        (* Constant: '<S391>/Constant4' incorporates:
         *  Constant: '<S391>/Constant'
         *  Constant: '<S391>/Constant1'
         *  Constant: '<S391>/Constant2'
         *  Constant: '<S391>/Constant3' *)
        i3_Chart_Hysteresis_LowActive(ssMethodType := SS_INITIALIZE, sSignal := AI_DCHV_Plus_FB, boInitial_Value := FALSE, boValue_Activated := TRUE, boValue_Deactivated := FALSE, sLB := 5000.0, b_sUB := 10000.0);
        boOutput := i3_Chart_Hysteresis_LowActive.boOutput;
        (* SystemInitialize for Atomic SubSystem: '<Root>/ChiefMaster' *)
        (* SystemInitialize for Chart: '<S23>/Chart_DCPlus_Status' *)
        temporalCounter_i1_a(timerAction := 1, maxTime := 0);
        is_active_c54_ChiefMaster := 0;
        is_c54_ChiefMaster := ChiefMaster_IN_NO_ACTIVE_CHILD_f;
        (* SystemInitialize for Chart: '<S13>/delay1' *)
        temporalCounter_i1_h(timerAction := 1, maxTime := 0);
        is_active_c51_ChiefMaster := 0;
        is_c51_ChiefMaster := ChiefMaster_IN_NO_ACTIVE_CHILD_f;
        (* End of SystemInitialize for SubSystem: '<Root>/ChiefMaster' *)
        i0_InsulationMonitoringReq(ssMethodType := SS_INITIALIZE, IT_boUDC_KL15_D := rtb_IT_boUDC_KL15_D, IT_boUDC_KL15_C := rtb_IT_boUDC_KL15_C, IT_boBMS_HV_ON_BB := rtb_IT_boBMS_HV_ON_BB, IT_u8BMS_BB_No_MaxVoltage := rtb_Switch_a, IT_u8BMS_BB_No_MinVoltage := rtb_Switch2_k, IT_boBMS_SDError_BB1 := rtb_IT_boBMS_SDError_BB1, IT_boBMS_SDError_BB2 := rtb_IT_boBMS_SDError_BB1, IT_boBMS_SDError_BB3 := rtb_IT_boBMS_SDError_BB1, IT_boBMS_InsulationReadyOK_B1 := rtb_IT_boBMS_SDError_BB1, IT_boBMS_InsulationReadyOK_B2 := rtb_IT_boBMS_SDError_BB1, IT_boBMS_InsulationReadyOK_B3 := rtb_IT_boBMS_SDError_BB1, IT_boBMS_IMD_Active_BB1 := rtb_IT_boBMS_SDError_BB1, IT_boBMS_IMD_Active_BB2 := rtb_IT_boBMS_SDError_BB1, IT_boBMS_IMD_Active_BB3 := rtb_IT_boBMS_SDError_BB1, IT_boBMS_HV_REL_ON_BB1 := rtb_IT_boBMS_SDError_BB1, IT_boBMS_HV_REL_ON_BB2 := rtb_IT_boBMS_SDError_BB1, IT_boBMS_HV_REL_ON_BB3 := rtb_IT_boBMS_SDError_BB1, IT_sBMS_Batt1_Availability := DINT_TO_LREAL(rtb_UnitDelay5), IT_sBMS_Batt2_Availability := DINT_TO_LREAL(rtb_UnitDelay5), IT_sBMS_Batt3_Availability := DINT_TO_LREAL(rtb_UnitDelay5), IT_boUDC_EV_IsolationMeasurementRequest := rtb_IT_boUDC_EV_IsolationMeasurementRequest, FL_boSS_System_SD := System_Error, FL_boSS_System_ESD := rtb_Delay_j);
        rtb_IT_boChargeStop_Button := i0_InsulationMonitoringReq.FL_boREQ_IMD_ON_BB1;
        rtb_UnitDelay1_d := i0_InsulationMonitoringReq.FL_boREQ_IMD_ON_BB2;
        rtb_Out_bl := i0_InsulationMonitoringReq.FL_boREQ_IMD_ON_BB3;
        rtb_IMD_State_g := i0_InsulationMonitoringReq.FL_u8_IMD_State_BB1;
        rtb_System_SD_ErrorCode := i0_InsulationMonitoringReq.FL_u8_IMD_State_BB2;
        rtb_IMD_State := i0_InsulationMonitoringReq.FL_u8_IMD_State_BB3;
        (* Constant: '<S81>/Constant' *)
        i0_Chart_jj(ssMethodType := SS_INITIALIZE, In := ContactorState_f, b_n := 5.0);
        rtb_IT_boUDC_EV_IsolationMeasurementRequest := i0_Chart_jj.Out;
        i0_Chart1(ssMethodType := SS_INITIALIZE, In := rtb_IT_boBMS_SDError_BB1);
        rtb_Out_ap := i0_Chart1.Out;
        (* Constant: '<S82>/Constant' *)
        i1_Chart_jj(ssMethodType := SS_INITIALIZE, In := ContactorState, b_n := 5.0);
        rtb_IT_boUDC_EV_IsolationMeasurementRequest := i1_Chart_jj.Out;
        i1_Chart1(ssMethodType := SS_INITIALIZE, In := rtb_IT_boBMS_SDError_BB1);
        rtb_Out_ap := i1_Chart1.Out;
        i0_Chart_lg(ssMethodType := SS_INITIALIZE, Error := rtb_IT_boBMS_SDError_BB1, KL15_reset := rtb_IT_boBMS_SDError_BB1);
        rtb_IT_boUDC_EV_IsolationMeasurementRequest := i0_Chart_lg.SW_Reset;
        i0_Chart1_l(ssMethodType := SS_INITIALIZE, SW_Reset := rtb_IT_boUDC_EV_IsolationMeasurementRequest, KL_15_reset_CM := rtb_IT_boBMS_SDError_BB1);
        Count_k := i0_Chart1_l.Count;
        i1_Chart_lg(ssMethodType := SS_INITIALIZE, Error := rtb_IT_boBMS_SDError_BB1, KL15_reset := rtb_IT_boBMS_SDError_BB1);
        rtb_IT_boUDC_EV_IsolationMeasurementRequest := i1_Chart_lg.SW_Reset;
        i1_Chart1_l(ssMethodType := SS_INITIALIZE, SW_Reset := rtb_IT_boUDC_EV_IsolationMeasurementRequest, KL_15_reset_CM := rtb_IT_boBMS_SDError_BB1);
        Count_k := i1_Chart1_l.Count;
        i2_Chart_lg(ssMethodType := SS_INITIALIZE, Error := rtb_IT_boBMS_SDError_BB1, KL15_reset := rtb_IT_boBMS_SDError_BB1);
        rtb_IT_boUDC_EV_IsolationMeasurementRequest := i2_Chart_lg.SW_Reset;
        i2_Chart1_l(ssMethodType := SS_INITIALIZE, SW_Reset := rtb_IT_boUDC_EV_IsolationMeasurementRequest, KL_15_reset_CM := rtb_IT_boBMS_SDError_BB1);
        Count_k := i2_Chart1_l.Count;
        (* Constant: '<S86>/Constant' *)
        i2_Chart_jj(ssMethodType := SS_INITIALIZE, In := ContactorState_i, b_n := 5.0);
        rtb_IT_boUDC_EV_IsolationMeasurementRequest := i2_Chart_jj.Out;
        i2_Chart1(ssMethodType := SS_INITIALIZE, In := rtb_IT_boBMS_SDError_BB1);
        rtb_Out_ap := i2_Chart1.Out;
        i0_CMState(ssMethodType := SS_INITIALIZE, KL15 := rtb_IT_boBMS_SDError_BB1, KL15_AllBoxes := rtb_IT_boBMS_SDError_BB1, InsulationReadyOK := rtb_IT_boBMS_SDError_BB1, BattRelay_Closed := rtb_IT_boBMS_SDError_BB1, IMD_Available := rtb_IT_boBMS_SDError_BB1, BattRelay_Close_Req := rtb_IT_boBMS_SDError_BB1, REQ_IMD_ON := rtb_IT_boBMS_SDError_BB1, FL_boREQ_MainHV_ON_MINUS := rtb_IT_boBMS_SDError_BB1, MainHV_Plus_Status := DINT_TO_LREAL(rtb_UnitDelay5), ShutdownError := rtb_IT_boBMS_SDError_BB1);
        CMState_e2 := i0_CMState.FL_u8SS_ChiefMaster_State;
        (* Outport: '<Root>/DO_boEMSRET_BB1_1' *)
        i0_EMSRET_Power(ssMethodType := SS_INITIALIZE, ESD := rtb_Delay_j, HVILNOK := rtb_FL_boSS_HVIL_NOK, b_Reset := rtb_FL_boKL15_Reset);
        DO_boEMSRET_BB1_1 := i0_EMSRET_Power.FL_boSS_EMSRET_POWER;
        (* SystemInitialize for Atomic SubSystem: '<Root>/ChiefMaster' *)
        (* SystemInitialize for Chart: '<S108>/Chart' *)
        temporalCounter_i1(timerAction := 1, maxTime := 0);
        is_active_c49_ChiefMaster := 0;
        is_c49_ChiefMaster := ChiefMaster_IN_NO_ACTIVE_CHILD_f;
        (* End of SystemInitialize for SubSystem: '<Root>/ChiefMaster' *)
        

        (* ConstCode for Atomic SubSystem: '<Root>/ChiefMaster' *)
        (* ConstCode for ArithShift: '<S823>/Shift Arithmetic' incorporates:
         *  Constant: '<S803>/Constant' *)
        ShiftArithmetic := 0;
        (* ConstCode for ArithShift: '<S823>/Shift Arithmetic2' incorporates:
         *  Constant: '<S803>/Constant' *)
        ShiftArithmetic2 := 0;
        (* ConstCode for ArithShift: '<S823>/Shift Arithmetic4' incorporates:
         *  Constant: '<S803>/Constant' *)
        ShiftArithmetic4 := 0;
        (* ConstCode for ArithShift: '<S823>/Shift Arithmetic5' incorporates:
         *  Constant: '<S803>/Constant' *)
        ShiftArithmetic5 := 0;
        (* ConstCode for ArithShift: '<S823>/Shift Arithmetic6' incorporates:
         *  Constant: '<S803>/Constant' *)
        ShiftArithmetic6 := 0;
        (* ConstCode for ArithShift: '<S824>/Shift Arithmetic' incorporates:
         *  Constant: '<S803>/Constant2' *)
        ShiftArithmetic_n := 0;
        (* ConstCode for ArithShift: '<S824>/Shift Arithmetic2' incorporates:
         *  Constant: '<S803>/Constant2' *)
        ShiftArithmetic2_c := 0;
        (* ConstCode for ArithShift: '<S824>/Shift Arithmetic3' incorporates:
         *  Constant: '<S803>/Constant2' *)
        ShiftArithmetic3 := 0;
        (* ConstCode for ArithShift: '<S824>/Shift Arithmetic4' incorporates:
         *  Constant: '<S803>/Constant2' *)
        ShiftArithmetic4_h := 0;
        (* ConstCode for ArithShift: '<S824>/Shift Arithmetic5' incorporates:
         *  Constant: '<S803>/Constant2' *)
        ShiftArithmetic5_j := 0;
        (* ConstCode for ArithShift: '<S824>/Shift Arithmetic6' incorporates:
         *  Constant: '<S803>/Constant2' *)
        ShiftArithmetic6_a := 0;
        (* ConstCode for ArithShift: '<S825>/Shift Arithmetic6' incorporates:
         *  Constant: '<S803>/Constant' *)
        ShiftArithmetic6_f := 0;
        (* ConstCode for ArithShift: '<S860>/Shift Arithmetic2' incorporates:
         *  Constant: '<S804>/Constant4' *)
        ShiftArithmetic2_o := 0;
        (* ConstCode for ArithShift: '<S860>/Shift Arithmetic5' incorporates:
         *  Constant: '<S804>/Constant4' *)
        ShiftArithmetic5_h := 0;
        (* ConstCode for ArithShift: '<S898>/Shift Arithmetic2' incorporates:
         *  Constant: '<S807>/Constant4' *)
        ShiftArithmetic2_n := 0;
        (* ConstCode for ArithShift: '<S898>/Shift Arithmetic5' incorporates:
         *  Constant: '<S807>/Constant4' *)
        ShiftArithmetic5_jh := 0;
        (* ConstCode for ArithShift: '<S937>/Shift Arithmetic2' incorporates:
         *  Constant: '<S810>/Constant4' *)
        ShiftArithmetic2_h := 0;
        (* ConstCode for ArithShift: '<S937>/Shift Arithmetic5' incorporates:
         *  Constant: '<S810>/Constant4' *)
        ShiftArithmetic5_f := 0;
        (* ConstCode for ArithShift: '<S973>/Shift Arithmetic' incorporates:
         *  Constant: '<S813>/Constant' *)
        ShiftArithmetic_m := 0;
        (* ConstCode for ArithShift: '<S973>/Shift Arithmetic2' incorporates:
         *  Constant: '<S813>/Constant' *)
        ShiftArithmetic2_k := 0;
        (* ConstCode for ArithShift: '<S973>/Shift Arithmetic4' incorporates:
         *  Constant: '<S813>/Constant' *)
        ShiftArithmetic4_m := 0;
        (* ConstCode for ArithShift: '<S981>/Shift Arithmetic5' incorporates:
         *  Constant: '<S814>/Constant1' *)
        ShiftArithmetic5_k := 0;
        (* ConstCode for ArithShift: '<S981>/Shift Arithmetic6' incorporates:
         *  Constant: '<S814>/Constant1' *)
        ShiftArithmetic6_i := 0;
        (* ConstCode for ArithShift: '<S982>/Shift Arithmetic2' incorporates:
         *  Constant: '<S814>/Constant3' *)
        ShiftArithmetic2_p := 0;
        (* ConstCode for ArithShift: '<S982>/Shift Arithmetic3' incorporates:
         *  Constant: '<S814>/Constant3' *)
        ShiftArithmetic3_k := 0;
        (* ConstCode for ArithShift: '<S982>/Shift Arithmetic4' incorporates:
         *  Constant: '<S814>/Constant3' *)
        ShiftArithmetic4_a := 0;
        (* ConstCode for ArithShift: '<S982>/Shift Arithmetic5' incorporates:
         *  Constant: '<S814>/Constant3' *)
        ShiftArithmetic5_a := 0;
        (* ConstCode for ArithShift: '<S982>/Shift Arithmetic6' incorporates:
         *  Constant: '<S814>/Constant3' *)
        ShiftArithmetic6_m := 0;
        (* ConstCode for ArithShift: '<S991>/Shift Arithmetic2' incorporates:
         *  Constant: '<S815>/Constant4' *)
        ShiftArithmetic2_d := 0;
        (* ConstCode for ArithShift: '<S991>/Shift Arithmetic4' incorporates:
         *  Constant: '<S815>/Constant4' *)
        ShiftArithmetic4_n := 0;
        (* ConstCode for ArithShift: '<S991>/Shift Arithmetic6' incorporates:
         *  Constant: '<S815>/Constant4' *)
        ShiftArithmetic6_h := 0;
        (* ConstCode for ArithShift: '<S992>/Shift Arithmetic2' incorporates:
         *  Constant: '<S815>/Constant4' *)
        ShiftArithmetic2_b := 0;
        (* ConstCode for ArithShift: '<S992>/Shift Arithmetic3' incorporates:
         *  Constant: '<S815>/Constant4' *)
        ShiftArithmetic3_o := 0;
        (* ConstCode for ArithShift: '<S992>/Shift Arithmetic5' incorporates:
         *  Constant: '<S815>/Constant4' *)
        ShiftArithmetic5_a2 := 0;
        (* ConstCode for ArithShift: '<S992>/Shift Arithmetic6' incorporates:
         *  Constant: '<S815>/Constant4' *)
        ShiftArithmetic6_n := 0;
        (* ConstCode for ArithShift: '<S993>/Shift Arithmetic' incorporates:
         *  Constant: '<S815>/Constant1' *)
        ShiftArithmetic_h := 0;
        (* ConstCode for ArithShift: '<S993>/Shift Arithmetic1' incorporates:
         *  Constant: '<S815>/Constant1' *)
        ShiftArithmetic1 := 0;
        (* ConstCode for ArithShift: '<S993>/Shift Arithmetic3' incorporates:
         *  Constant: '<S815>/Constant1' *)
        ShiftArithmetic3_e := 0;
        (* ConstCode for ArithShift: '<S993>/Shift Arithmetic4' incorporates:
         *  Constant: '<S815>/Constant1' *)
        ShiftArithmetic4_ap := 0;
        (* ConstCode for ArithShift: '<S993>/Shift Arithmetic5' incorporates:
         *  Constant: '<S815>/Constant1' *)
        ShiftArithmetic5_i := 0;
        (* ConstCode for ArithShift: '<S993>/Shift Arithmetic6' incorporates:
         *  Constant: '<S815>/Constant1' *)
        ShiftArithmetic6_k := 0;
        (* ConstCode for DataTypeConversion: '<S1020>/Data Type Conversion1' incorporates:
         *  Constant: '<S1017>/Constant15' *)
        DataTypeConversion1 := 0;
        (* ConstCode for DataTypeConversion: '<S1020>/Data Type Conversion2' incorporates:
         *  Constant: '<S1017>/Constant15' *)
        DataTypeConversion2 := 0;
        (* ConstCode for DataTypeConversion: '<S1020>/Data Type Conversion4' incorporates:
         *  Constant: '<S1017>/Constant15' *)
        DataTypeConversion4 := 0;
        (* ConstCode for DataTypeConversion: '<S1020>/Data Type Conversion5' incorporates:
         *  Constant: '<S1017>/Constant15' *)
        DataTypeConversion5 := 0;
        (* ConstCode for DataTypeConversion: '<S1020>/Data Type Conversion6' incorporates:
         *  Constant: '<S1017>/Constant15' *)
        DataTypeConversion6 := 0;
        (* ConstCode for DataTypeConversion: '<S1020>/Data Type Conversion7' incorporates:
         *  Constant: '<S1017>/Constant15' *)
        DataTypeConversion7 := 0;
        (* ConstCode for ArithShift: '<S1020>/Shift Arithmetic1' incorporates:
         *  DataTypeConversion: '<S1020>/Data Type Conversion1' *)
        ShiftArithmetic1_n := BYTE_TO_USINT(SHL(USINT_TO_BYTE(DataTypeConversion1), 2));
        (* ConstCode for ArithShift: '<S1020>/Shift Arithmetic2' incorporates:
         *  DataTypeConversion: '<S1020>/Data Type Conversion2' *)
        ShiftArithmetic2_ot := BYTE_TO_USINT(SHL(USINT_TO_BYTE(DataTypeConversion2), 3));
        (* ConstCode for ArithShift: '<S1020>/Shift Arithmetic3' incorporates:
         *  DataTypeConversion: '<S1020>/Data Type Conversion4' *)
        ShiftArithmetic3_oe := BYTE_TO_USINT(SHL(USINT_TO_BYTE(DataTypeConversion4), 4));
        (* ConstCode for ArithShift: '<S1020>/Shift Arithmetic4' incorporates:
         *  DataTypeConversion: '<S1020>/Data Type Conversion5' *)
        ShiftArithmetic4_d := BYTE_TO_USINT(SHL(USINT_TO_BYTE(DataTypeConversion5), 5));
        (* ConstCode for ArithShift: '<S1020>/Shift Arithmetic5' incorporates:
         *  DataTypeConversion: '<S1020>/Data Type Conversion6' *)
        ShiftArithmetic5_ke := BYTE_TO_USINT(SHL(USINT_TO_BYTE(DataTypeConversion6), 6));
        (* ConstCode for ArithShift: '<S1020>/Shift Arithmetic6' incorporates:
         *  DataTypeConversion: '<S1020>/Data Type Conversion7' *)
        ShiftArithmetic6_kx := BYTE_TO_USINT(SHL(USINT_TO_BYTE(DataTypeConversion7), 7));
        (* ConstCode for DataTypeConversion: '<S1021>/Data Type Conversion1' incorporates:
         *  Constant: '<S1018>/Constant1' *)
        DataTypeConversion1_l := 0;
        (* ConstCode for DataTypeConversion: '<S1021>/Data Type Conversion2' incorporates:
         *  Constant: '<S1018>/Constant1' *)
        DataTypeConversion2_b := 0;
        (* ConstCode for DataTypeConversion: '<S1021>/Data Type Conversion4' incorporates:
         *  Constant: '<S1018>/Constant1' *)
        DataTypeConversion4_l := 0;
        (* ConstCode for DataTypeConversion: '<S1021>/Data Type Conversion5' incorporates:
         *  Constant: '<S1018>/Constant1' *)
        DataTypeConversion5_k := 0;
        (* ConstCode for DataTypeConversion: '<S1021>/Data Type Conversion6' incorporates:
         *  Constant: '<S1018>/Constant1' *)
        DataTypeConversion6_e := 0;
        (* ConstCode for DataTypeConversion: '<S1021>/Data Type Conversion7' incorporates:
         *  Constant: '<S1018>/Constant1' *)
        DataTypeConversion7_p := 0;
        (* ConstCode for ArithShift: '<S1021>/Shift Arithmetic1' incorporates:
         *  DataTypeConversion: '<S1021>/Data Type Conversion1' *)
        ShiftArithmetic1_nm := BYTE_TO_USINT(SHL(USINT_TO_BYTE(DataTypeConversion1_l), 2));
        (* ConstCode for ArithShift: '<S1021>/Shift Arithmetic2' incorporates:
         *  DataTypeConversion: '<S1021>/Data Type Conversion2' *)
        ShiftArithmetic2_e := BYTE_TO_USINT(SHL(USINT_TO_BYTE(DataTypeConversion2_b), 3));
        (* ConstCode for ArithShift: '<S1021>/Shift Arithmetic3' incorporates:
         *  DataTypeConversion: '<S1021>/Data Type Conversion4' *)
        ShiftArithmetic3_o0 := BYTE_TO_USINT(SHL(USINT_TO_BYTE(DataTypeConversion4_l), 4));
        (* ConstCode for ArithShift: '<S1021>/Shift Arithmetic4' incorporates:
         *  DataTypeConversion: '<S1021>/Data Type Conversion5' *)
        ShiftArithmetic4_b := BYTE_TO_USINT(SHL(USINT_TO_BYTE(DataTypeConversion5_k), 5));
        (* ConstCode for ArithShift: '<S1021>/Shift Arithmetic5' incorporates:
         *  DataTypeConversion: '<S1021>/Data Type Conversion6' *)
        ShiftArithmetic5_hi := BYTE_TO_USINT(SHL(USINT_TO_BYTE(DataTypeConversion6_e), 6));
        (* ConstCode for ArithShift: '<S1021>/Shift Arithmetic6' incorporates:
         *  DataTypeConversion: '<S1021>/Data Type Conversion7' *)
        ShiftArithmetic6_kxt := BYTE_TO_USINT(SHL(USINT_TO_BYTE(DataTypeConversion7_p), 7));
        (* ConstCode for DataTypeConversion: '<S1022>/Data Type Conversion1' incorporates:
         *  Constant: '<S1019>/Constant2' *)
        DataTypeConversion1_o := 0;
        (* ConstCode for DataTypeConversion: '<S1022>/Data Type Conversion2' incorporates:
         *  Constant: '<S1019>/Constant2' *)
        DataTypeConversion2_o := 0;
        (* ConstCode for DataTypeConversion: '<S1022>/Data Type Conversion4' incorporates:
         *  Constant: '<S1019>/Constant2' *)
        DataTypeConversion4_i := 0;
        (* ConstCode for DataTypeConversion: '<S1022>/Data Type Conversion5' incorporates:
         *  Constant: '<S1019>/Constant2' *)
        DataTypeConversion5_n := 0;
        (* ConstCode for DataTypeConversion: '<S1022>/Data Type Conversion6' incorporates:
         *  Constant: '<S1019>/Constant2' *)
        DataTypeConversion6_k := 0;
        (* ConstCode for DataTypeConversion: '<S1022>/Data Type Conversion7' incorporates:
         *  Constant: '<S1019>/Constant2' *)
        DataTypeConversion7_pe := 0;
        (* ConstCode for ArithShift: '<S1022>/Shift Arithmetic1' incorporates:
         *  DataTypeConversion: '<S1022>/Data Type Conversion1' *)
        ShiftArithmetic1_nx := BYTE_TO_USINT(SHL(USINT_TO_BYTE(DataTypeConversion1_o), 2));
        (* ConstCode for ArithShift: '<S1022>/Shift Arithmetic2' incorporates:
         *  DataTypeConversion: '<S1022>/Data Type Conversion2' *)
        ShiftArithmetic2_m := BYTE_TO_USINT(SHL(USINT_TO_BYTE(DataTypeConversion2_o), 3));
        (* ConstCode for ArithShift: '<S1022>/Shift Arithmetic3' incorporates:
         *  DataTypeConversion: '<S1022>/Data Type Conversion4' *)
        ShiftArithmetic3_a := BYTE_TO_USINT(SHL(USINT_TO_BYTE(DataTypeConversion4_i), 4));
        (* ConstCode for ArithShift: '<S1022>/Shift Arithmetic4' incorporates:
         *  DataTypeConversion: '<S1022>/Data Type Conversion5' *)
        ShiftArithmetic4_p := BYTE_TO_USINT(SHL(USINT_TO_BYTE(DataTypeConversion5_n), 5));
        (* ConstCode for ArithShift: '<S1022>/Shift Arithmetic5' incorporates:
         *  DataTypeConversion: '<S1022>/Data Type Conversion6' *)
        ShiftArithmetic5_b := BYTE_TO_USINT(SHL(USINT_TO_BYTE(DataTypeConversion6_k), 6));
        (* ConstCode for ArithShift: '<S1022>/Shift Arithmetic6' incorporates:
         *  DataTypeConversion: '<S1022>/Data Type Conversion7' *)
        ShiftArithmetic6_b := BYTE_TO_USINT(SHL(USINT_TO_BYTE(DataTypeConversion7_pe), 7));
        (* ConstCode for DataTypeConversion: '<S1026>/Extract Desired Bits' incorporates:
         *  Constant: '<S1023>/Constant4' *)
        ExtractDesiredBits := 0;
        (* ConstCode for DataTypeConversion: '<S1028>/Extract Desired Bits' incorporates:
         *  Constant: '<S1023>/Constant5' *)
        ExtractDesiredBits_m := 1;
        (* ConstCode for DataTypeConversion: '<S1031>/Data Type Conversion3' incorporates:
         *  DataTypeConversion: '<S1026>/Extract Desired Bits' *)
        DataTypeConversion3 := ExtractDesiredBits;
        (* ConstCode for DataTypeConversion: '<S1031>/Data Type Conversion6' incorporates:
         *  DataTypeConversion: '<S1028>/Extract Desired Bits' *)
        DataTypeConversion6_h := ExtractDesiredBits_m;
        (* ConstCode for ArithShift: '<S1031>/Shift Arithmetic' incorporates:
         *  Constant: '<S1023>/Constant1' *)
        ShiftArithmetic_k := 0;
        (* ConstCode for ArithShift: '<S1031>/Shift Arithmetic2' incorporates:
         *  Constant: '<S1023>/Constant2' *)
        ShiftArithmetic2_f := 0;
        (* ConstCode for ArithShift: '<S1031>/Shift Arithmetic3' incorporates:
         *  Constant: '<S1023>/Constant2' *)
        ShiftArithmetic3_h := 0;
        (* ConstCode for ArithShift: '<S1031>/Shift Arithmetic4' incorporates:
         *  Constant: '<S1023>/Constant2' *)
        ShiftArithmetic4_l := 0;
        (* ConstCode for ArithShift: '<S1031>/Shift Arithmetic5' incorporates:
         *  DataTypeConversion: '<S1031>/Data Type Conversion6' *)
        ShiftArithmetic5_m := BYTE_TO_USINT(SHL(USINT_TO_BYTE(DataTypeConversion6_h), 6));
        (* ConstCode for ArithShift: '<S1031>/Shift Arithmetic6' incorporates:
         *  Constant: '<S1023>/Constant3' *)
        ShiftArithmetic6_ap := 0;
        (* ConstCode for DataTypeConversion: '<S1032>/Extract Desired Bits' incorporates:
         *  Constant: '<S1024>/Constant4' *)
        ExtractDesiredBits_n := 0;
        (* ConstCode for DataTypeConversion: '<S1034>/Extract Desired Bits' incorporates:
         *  Constant: '<S1024>/Constant5' *)
        ExtractDesiredBits_b := 1;
        (* ConstCode for DataTypeConversion: '<S1037>/Data Type Conversion3' incorporates:
         *  DataTypeConversion: '<S1032>/Extract Desired Bits' *)
        DataTypeConversion3_d := ExtractDesiredBits_n;
        (* ConstCode for DataTypeConversion: '<S1037>/Data Type Conversion6' incorporates:
         *  DataTypeConversion: '<S1034>/Extract Desired Bits' *)
        DataTypeConversion6_p := ExtractDesiredBits_b;
        (* ConstCode for ArithShift: '<S1037>/Shift Arithmetic' incorporates:
         *  Constant: '<S1024>/Constant1' *)
        ShiftArithmetic_a := 0;
        (* ConstCode for ArithShift: '<S1037>/Shift Arithmetic2' incorporates:
         *  Constant: '<S1024>/Constant2' *)
        ShiftArithmetic2_fl := 0;
        (* ConstCode for ArithShift: '<S1037>/Shift Arithmetic3' incorporates:
         *  Constant: '<S1024>/Constant2' *)
        ShiftArithmetic3_l := 0;
        (* ConstCode for ArithShift: '<S1037>/Shift Arithmetic4' incorporates:
         *  Constant: '<S1024>/Constant2' *)
        ShiftArithmetic4_f := 0;
        (* ConstCode for ArithShift: '<S1037>/Shift Arithmetic5' incorporates:
         *  DataTypeConversion: '<S1037>/Data Type Conversion6' *)
        ShiftArithmetic5_k0 := BYTE_TO_USINT(SHL(USINT_TO_BYTE(DataTypeConversion6_p), 6));
        (* ConstCode for ArithShift: '<S1037>/Shift Arithmetic6' incorporates:
         *  Constant: '<S1024>/Constant3' *)
        ShiftArithmetic6_o := 0;
        (* ConstCode for DataTypeConversion: '<S1038>/Extract Desired Bits' incorporates:
         *  Constant: '<S1025>/Constant4' *)
        ExtractDesiredBits_m1 := 0;
        (* ConstCode for DataTypeConversion: '<S1040>/Extract Desired Bits' incorporates:
         *  Constant: '<S1025>/Constant5' *)
        ExtractDesiredBits_p := 1;
        (* ConstCode for DataTypeConversion: '<S1043>/Data Type Conversion3' incorporates:
         *  DataTypeConversion: '<S1038>/Extract Desired Bits' *)
        DataTypeConversion3_l := ExtractDesiredBits_m1;
        (* ConstCode for DataTypeConversion: '<S1043>/Data Type Conversion6' incorporates:
         *  DataTypeConversion: '<S1040>/Extract Desired Bits' *)
        DataTypeConversion6_l := ExtractDesiredBits_p;
        (* ConstCode for ArithShift: '<S1043>/Shift Arithmetic' incorporates:
         *  Constant: '<S1025>/Constant1' *)
        ShiftArithmetic_p := 0;
        (* ConstCode for ArithShift: '<S1043>/Shift Arithmetic2' incorporates:
         *  Constant: '<S1025>/Constant2' *)
        ShiftArithmetic2_g := 0;
        (* ConstCode for ArithShift: '<S1043>/Shift Arithmetic3' incorporates:
         *  Constant: '<S1025>/Constant2' *)
        ShiftArithmetic3_c := 0;
        (* ConstCode for ArithShift: '<S1043>/Shift Arithmetic4' incorporates:
         *  Constant: '<S1025>/Constant2' *)
        ShiftArithmetic4_db := 0;
        (* ConstCode for ArithShift: '<S1043>/Shift Arithmetic5' incorporates:
         *  DataTypeConversion: '<S1043>/Data Type Conversion6' *)
        ShiftArithmetic5_c := BYTE_TO_USINT(SHL(USINT_TO_BYTE(DataTypeConversion6_l), 6));
        (* ConstCode for ArithShift: '<S1043>/Shift Arithmetic6' incorporates:
         *  Constant: '<S1025>/Constant3' *)
        ShiftArithmetic6_mw := 0;
        (* End of ConstCode for SubSystem: '<Root>/ChiefMaster' *)
    SS_STEP: 
        (* Outputs for Atomic SubSystem: '<Root>/ChiefMaster' *)
        (* Outputs for Enabled SubSystem: '<S195>/Subsystem1' incorporates:
         *  EnablePort: '<S664>/Timeout' *)
        (* Logic: '<S195>/NOT' *)

        IF  NOT C_UDC_Msg1_Timeout THEN 

            IF  NOT Subsystem1_MODE THEN 
                Subsystem1_MODE := TRUE;
            END_IF;

            (* DataTypeConversion: '<S664>/Data Type Conversion2' incorporates:
             *  DataTypeConversion: '<S666>/Extract Desired Bits' *)
            IP_boSafeToShutdown := DWORD_TO_UDINT(UDINT_TO_DWORD(USINT_TO_UDINT(C_UDC_Msg1[0])) AND 1) <> 0;
            (* DataTypeConversion: '<S664>/Data Type Conversion3' incorporates:
             *  DataTypeConversion: '<S667>/Extract Desired Bits' *)
            IP_boKL15_D := DWORD_TO_UDINT(UDINT_TO_DWORD(DINT_TO_UDINT(DWORD_TO_DINT(SHR(DINT_TO_DWORD(USINT_TO_DINT(C_UDC_Msg1[0])), 1)))) AND 1) <> 0;
            (* DataTypeConversion: '<S664>/Data Type Conversion4' incorporates:
             *  DataTypeConversion: '<S668>/Extract Desired Bits' *)
            IP_boKL15_C := DWORD_TO_UDINT(UDINT_TO_DWORD(DINT_TO_UDINT(DWORD_TO_DINT(SHR(DINT_TO_DWORD(USINT_TO_DINT(C_UDC_Msg1[0])), 2)))) AND 1) <> 0;
            (* DataTypeConversion: '<S664>/Data Type Conversion5' incorporates:
             *  DataTypeConversion: '<S669>/Extract Desired Bits' *)
            IP_boEVDisconnectingDevice := DWORD_TO_UDINT(UDINT_TO_DWORD(DINT_TO_UDINT(DWORD_TO_DINT(SHR(DINT_TO_DWORD(USINT_TO_DINT(C_UDC_Msg1[0])), 3)))) AND 1) <> 0;
            (* DataTypeConversion: '<S664>/Data Type Conversion7' incorporates:
             *  DataTypeConversion: '<S671>/Extract Desired Bits' *)
            IP_boChargeStop_Button := DWORD_TO_UDINT(UDINT_TO_DWORD(DINT_TO_UDINT(DWORD_TO_DINT(SHR(DINT_TO_DWORD(USINT_TO_DINT(C_UDC_Msg1[0])), 5)))) AND 1) <> 0;
            (* SignalConversion: '<S664>/TmpBufferAtConstantOutport1' incorporates:
             *  Constant: '<S664>/Constant' *)
            IP_boEV_IsolationMeasurementRequest := TRUE;
        ELSIF Subsystem1_MODE THEN 
            (* Disable for DataTypeConversion: '<S664>/Data Type Conversion2' incorporates:
             *  Outport: '<S664>/TTC_Status_Databus' *)
            IP_boSafeToShutdown := FALSE;
            (* Disable for DataTypeConversion: '<S664>/Data Type Conversion3' incorporates:
             *  Outport: '<S664>/TTC_Status_Databus' *)
            IP_boKL15_D := FALSE;
            (* Disable for DataTypeConversion: '<S664>/Data Type Conversion4' incorporates:
             *  Outport: '<S664>/TTC_Status_Databus' *)
            IP_boKL15_C := FALSE;
            (* Disable for DataTypeConversion: '<S664>/Data Type Conversion5' incorporates:
             *  Outport: '<S664>/TTC_Status_Databus' *)
            IP_boEVDisconnectingDevice := FALSE;
            (* Disable for SignalConversion: '<S664>/TmpBufferAtConstantOutport1' incorporates:
             *  Outport: '<S664>/TTC_Status_Databus' *)
            IP_boEV_IsolationMeasurementRequest := FALSE;
            (* Disable for DataTypeConversion: '<S664>/Data Type Conversion7' incorporates:
             *  Outport: '<S664>/TTC_Status_Databus' *)
            IP_boChargeStop_Button := FALSE;
            Subsystem1_MODE := FALSE;
        END_IF;

        (* End of Logic: '<S195>/NOT' *)
        (* End of Outputs for SubSystem: '<S195>/Subsystem1' *)
        

        (* SignalConversion: '<S678>/Signal Copy5' *)
        rtb_IT_boUDC_EV_IsolationMeasurementRequest := IP_boEV_IsolationMeasurementRequest;
        (* SignalConversion: '<S678>/Signal Copy6' *)
        rtb_IT_boChargeStop_Button := IP_boChargeStop_Button;
        (* End of Outputs for SubSystem: '<Root>/ChiefMaster' *)
        

        (* Constant: '<S387>/Constant4' incorporates:
         *  Constant: '<S387>/Constant'
         *  Constant: '<S387>/Constant1'
         *  Constant: '<S387>/Constant2'
         *  Constant: '<S387>/Constant3' *)
        i5_Chart_Hysteresis_HighActive(ssMethodType := SS_OUTPUT, sSignal := AI_KL15, boInitial_Value := FALSE, boValue_Activated := TRUE, boValue_Deactivated := FALSE, sLB := 18000.0, b_sUB := 22000.0);
        boOutput_c := i5_Chart_Hysteresis_HighActive.boOutput;
        (* Outputs for Atomic SubSystem: '<Root>/ChiefMaster' *)
        (* SignalConversion: '<S677>/Signal Copy' *)
        rtb_IT_boBMS_SDError_BB1 := boOutput_c;
        (* Logic: '<S55>/NOT1' incorporates:
         *  RelationalOperator: '<S61>/Compare'
         *  SignalConversion: '<S677>/Signal Copy' *)
        rtb_S_in :=  NOT boOutput_c;
        (* Logic: '<S56>/NOT' incorporates:
         *  Constant: '<S60>/Constant'
         *  Constant: '<S62>/Constant'
         *  Constant: '<S63>/Constant'
         *  Logic: '<S56>/OR'
         *  Logic: '<S56>/OR1'
         *  Logic: '<S56>/OR2'
         *  Outport: '<Root>/DO_KL15_BB1'
         *  RelationalOperator: '<S60>/Compare'
         *  RelationalOperator: '<S62>/Compare'
         *  RelationalOperator: '<S63>/Compare'
         *  UnitDelay: '<S10>/Unit Delay'
         *  UnitDelay: '<S10>/Unit Delay6' *)
        i0_Chart_m(ssMethodType := SS_OUTPUT, In := (( NOT rtb_S_in) AND (UnitDelay_DSTATE <> 1.0)) OR ((UnitDelay6_DSTATE <> 1.0) AND (UnitDelay6_DSTATE <> 3.0)), KL15_CM_Reset := rtb_S_in);
        DO_KL15_BB1 := i0_Chart_m.Out;
        (* RelationalOperator: '<S66>/Compare' incorporates:
         *  Logic: '<S55>/NOR'
         *  RelationalOperator: '<S71>/Compare' *)
        rtb_out_n :=  NOT rtb_IT_boBMS_SDError_BB1;
        (* Logic: '<S57>/NOT' incorporates:
         *  Constant: '<S65>/Constant'
         *  Constant: '<S67>/Constant'
         *  Constant: '<S68>/Constant'
         *  Logic: '<S57>/OR'
         *  Logic: '<S57>/OR1'
         *  Logic: '<S57>/OR2'
         *  Outport: '<Root>/DO_KL15_BB2'
         *  RelationalOperator: '<S65>/Compare'
         *  RelationalOperator: '<S66>/Compare'
         *  RelationalOperator: '<S67>/Compare'
         *  RelationalOperator: '<S68>/Compare'
         *  UnitDelay: '<S10>/Unit Delay1'
         *  UnitDelay: '<S10>/Unit Delay7' *)
        i1_Chart_m(ssMethodType := SS_OUTPUT, In := (( NOT rtb_out_n) AND (UnitDelay1_DSTATE <> 1.0)) OR ((UnitDelay7_DSTATE <> 1.0) AND (UnitDelay7_DSTATE <> 3.0)), KL15_CM_Reset := rtb_out_n);
        DO_KL15_BB2 := i1_Chart_m.Out;
        (* Logic: '<S58>/NOT' incorporates:
         *  Constant: '<S70>/Constant'
         *  Constant: '<S72>/Constant'
         *  Constant: '<S73>/Constant'
         *  Logic: '<S58>/OR'
         *  Logic: '<S58>/OR1'
         *  Logic: '<S58>/OR2'
         *  Outport: '<Root>/DO_KL15_BB3'
         *  RelationalOperator: '<S70>/Compare'
         *  RelationalOperator: '<S72>/Compare'
         *  RelationalOperator: '<S73>/Compare'
         *  UnitDelay: '<S10>/Unit Delay2'
         *  UnitDelay: '<S10>/Unit Delay8' *)
        i2_Chart_m(ssMethodType := SS_OUTPUT, In := (( NOT rtb_out_n) AND (UnitDelay2_DSTATE <> 1.0)) OR ((UnitDelay8_DSTATE <> 1.0) AND (UnitDelay8_DSTATE <> 3.0)), KL15_CM_Reset := rtb_out_n);
        DO_KL15_BB3 := i2_Chart_m.Out;
        (* Logic: '<S55>/AND' incorporates:
         *  Logic: '<S55>/NOT1'
         *  Logic: '<S55>/NOT2'
         *  Logic: '<S55>/NOT3'
         *  Logic: '<S55>/NOT4'
         *  Outport: '<Root>/DO_KL15_BB1'
         *  Outport: '<Root>/DO_KL15_BB2'
         *  Outport: '<Root>/DO_KL15_BB3' *)
        rtb_FL_boCMSleep := ((rtb_S_in AND ( NOT DO_KL15_BB1)) AND ( NOT DO_KL15_BB2)) AND ( NOT DO_KL15_BB3);
        (* SignalConversion: '<S678>/Signal Copy1' *)
        rtb_IT_boUDC_KL15_D := IP_boKL15_D;
        (* SignalConversion: '<S678>/Signal Copy2' *)
        rtb_IT_boUDC_KL15_C := IP_boKL15_C;
        (* Logic: '<S55>/AND6' incorporates:
         *  SignalConversion: '<S678>/Signal Copy1'
         *  SignalConversion: '<S678>/Signal Copy2' *)
        rtb_FL_boKL15_Disable := IP_boKL15_D = IP_boKL15_C;
        (* Switch: '<S431>/Switch' incorporates:
         *  Constant: '<S431>/Constant'
         *  Constant: '<S431>/Constant1'
         *  Logic: '<S431>/AND'
         *  Logic: '<S431>/NOT'
         *  Logic: '<S431>/NOT1'
         *  Logic: '<S431>/NOT2'
         *  Logic: '<S431>/NOT3'
         *  Logic: '<S431>/NOT4'
         *  Logic: '<S431>/NOT5'
         *  Logic: '<S431>/NOT6' *)

        IF (((((( NOT C_LB_Batt1_CellVoltage01_Timeout) AND ( NOT C_LB_Batt1_CellVoltage02_Timeout)) AND ( NOT C_LB_Batt1_CellTemperature_Timeout)) AND ( NOT C_LB_Batt1_InsulationMonitor_Timeout)) AND ( NOT C_LB_Batt1_Status01_Timeout)) AND ( NOT C_LB_Batt1_Status02_Timeout)) AND ( NOT C_LB_Batt1_Status03_Timeout) THEN 
            rtb_Switch2_d := TRUE;
            (* Switch: '<S675>/Switch1' incorporates:
             *  Constant: '<S431>/Constant'
             *  Constant: '<S675>/Constant6' *)
            rtb_S_in := TRUE;
        ELSE 
            rtb_Switch2_d := FALSE;
            (* Switch: '<S675>/Switch1' incorporates:
             *  Constant: '<S431>/Constant1'
             *  Constant: '<S675>/Constant7' *)
            rtb_S_in := FALSE;
        END_IF;

        (* End of Switch: '<S431>/Switch' *)
        

        (* Switch: '<S200>/Switch' incorporates:
         *  Logic: '<S200>/AND'
         *  Logic: '<S200>/NOT'
         *  Logic: '<S200>/NOT1'
         *  Logic: '<S200>/NOT2'
         *  Logic: '<S200>/NOT3'
         *  Logic: '<S200>/NOT4'
         *  Logic: '<S200>/NOT5' *)

        IF ((((( NOT C_Actia_Batt1_MyStatus_Timeout) AND ( NOT C_Actia_Batt1_Error_Timeout)) AND ( NOT C_Actia_Batt1_ADS_8_Timeout)) AND ( NOT C_Actia_Batt1_ADS_0_Timeout)) AND ( NOT C_Actia_Batt1_ADS_1_Timeout)) AND ( NOT C_Actia_Batt1_ADS_3_Timeout) THEN 
            (* Switch: '<S675>/Switch' incorporates:
             *  Constant: '<S675>/Constant3' *)
            rtb_IP_boBatt1_Actia_Availability := TRUE;
        ELSE 
            (* Switch: '<S675>/Switch' incorporates:
             *  Constant: '<S675>/Constant4' *)
            rtb_IP_boBatt1_Actia_Availability := FALSE;
        END_IF;

        (* End of Switch: '<S200>/Switch' *)
        (* End of Outputs for SubSystem: '<Root>/ChiefMaster' *)
        i0_ChartBatt1(ssMethodType := SS_OUTPUT, BattAvailable_LiBa := rtb_S_in, BattAvailable_Actia := rtb_IP_boBatt1_Actia_Availability);
        rtb_BattSelect_f := i0_ChartBatt1.BattSelect;
        (* Outputs for Atomic SubSystem: '<Root>/ChiefMaster' *)
        (* Sum: '<S208>/Add' incorporates:
         *  ArithShift: '<S207>/Shift Arithmetic'
         *  Constant: '<S206>/Constant'
         *  DataTypeConversion: '<S207>/Data Type Conversion'
         *  Product: '<S208>/Product'
         *  Sum: '<S207>/Add' *)
        rtb_Min := DINT_TO_REAL(DWORD_TO_DINT(SHL(DINT_TO_DWORD(USINT_TO_DINT(C_Actia_Batt1_ADS_3[2])), 8)) + USINT_TO_DINT(C_Actia_Batt1_ADS_3[1])) * 0.1;
        (* Sum: '<S498>/Add' incorporates:
         *  ArithShift: '<S497>/Shift Arithmetic'
         *  Constant: '<S493>/Constant'
         *  DataTypeConversion: '<S497>/Data Type Conversion'
         *  Product: '<S498>/Product'
         *  Sum: '<S497>/Add' *)
        rtb_Add_psl := DINT_TO_REAL(DWORD_TO_DINT(SHL(DINT_TO_DWORD(USINT_TO_DINT(C_LB_BMS_Status02_Msg[7])), 8)) + USINT_TO_DINT(C_LB_BMS_Status02_Msg[6])) * 0.1;
        (* Switch: '<S498>/Switch' incorporates:
         *  Constant: '<S493>/Constant3'
         *  Constant: '<S493>/Constant4'
         *  RelationalOperator: '<S498>/GreaterThan'
         *  Switch: '<S498>/Switch1' *)

        IF C_LB_Batt1_Status02_Timeout THEN 
            rtb_Add_psl := 0.0;
        ELSIF rtb_Add_psl > 6553.5 THEN 
            (* Switch: '<S498>/Switch1' incorporates:
             *  Constant: '<S493>/Constant4' *)
            rtb_Add_psl := 0.0;
        END_IF;

        (* End of Switch: '<S498>/Switch' *)
        

        (* MultiPortSwitch: '<S712>/Multiport Switch' incorporates:
         *  Constant: '<S712>/Constant' *)

        CASE TRUNC(rtb_BattSelect_f) OF
            1: 
                (* Switch: '<S208>/Switch' incorporates:
                 *  Constant: '<S206>/Constant3'
                 *  Constant: '<S206>/SafeValue_NA '
                 *  RelationalOperator: '<S208>/GreaterThan'
                 *  Switch: '<S208>/Switch1' *)

                IF C_Actia_Batt1_ADS_3_Timeout THEN 
                    rtb_Min := 0.0;
                ELSIF rtb_Min > 6553.5 THEN 
                    (* Switch: '<S208>/Switch1' incorporates:
                     *  Constant: '<S206>/SafeValue_Error' *)
                    rtb_Min := 0.0;
                END_IF;

                (* End of Switch: '<S208>/Switch' *)
            2: 
                rtb_Min := rtb_Add_psl;
            3: 
                rtb_Min := 0.0;
            ELSE
                rtb_Min := 0.0;
        END_CASE;

        (* End of MultiPortSwitch: '<S712>/Multiport Switch' *)
        

        (* Switch: '<S511>/Switch' incorporates:
         *  Constant: '<S511>/Constant'
         *  Constant: '<S511>/Constant1'
         *  Logic: '<S511>/AND'
         *  Logic: '<S511>/NOT'
         *  Logic: '<S511>/NOT1'
         *  Logic: '<S511>/NOT2'
         *  Logic: '<S511>/NOT3'
         *  Logic: '<S511>/NOT4'
         *  Logic: '<S511>/NOT5'
         *  Logic: '<S511>/NOT6' *)

        IF (((((( NOT C_LB_Batt2_CellVoltage01_Timeout) AND ( NOT C_LB_Batt2_CellVoltage02_Timeout)) AND ( NOT C_LB_Batt2_CellTemperature_Timeout)) AND ( NOT C_LB_Batt2_InsulationMonitor_Timeout)) AND ( NOT C_LB_Batt2_Status01_Timeout)) AND ( NOT C_LB_Batt2_Status02_Timeout)) AND ( NOT C_LB_Batt2_Status03_Timeout) THEN 
            rtb_Switch1_fj := TRUE;
            (* Switch: '<S675>/Switch3' incorporates:
             *  Constant: '<S511>/Constant'
             *  Constant: '<S675>/Constant5' *)
            rtb_S_in := TRUE;
        ELSE 
            rtb_Switch1_fj := FALSE;
            (* Switch: '<S675>/Switch3' incorporates:
             *  Constant: '<S511>/Constant1'
             *  Constant: '<S675>/Constant8' *)
            rtb_S_in := FALSE;
        END_IF;

        (* End of Switch: '<S511>/Switch' *)
        

        (* Switch: '<S261>/Switch' incorporates:
         *  Constant: '<S261>/Constant'
         *  Constant: '<S261>/Constant1'
         *  Logic: '<S261>/AND'
         *  Logic: '<S261>/NOT'
         *  Logic: '<S261>/NOT1'
         *  Logic: '<S261>/NOT2'
         *  Logic: '<S261>/NOT3'
         *  Logic: '<S261>/NOT4'
         *  Logic: '<S261>/NOT5' *)

        IF ((((( NOT C_Actia_Batt2_MyStatus_Timeout) AND ( NOT C_Actia_Batt2_Error_Timeout)) AND ( NOT C_Actia_Batt2_ADS_8_Timeout)) AND ( NOT C_Actia_Batt2_ADS_0_Timeout)) AND ( NOT C_Actia_Batt2_ADS_1_Timeout)) AND ( NOT C_Actia_Batt2_ADS_3_Timeout) THEN 
            rtb_UnitDelay5 := 1;
            (* Switch: '<S675>/Switch2' incorporates:
             *  Constant: '<S261>/Constant'
             *  Constant: '<S675>/Constant1' *)
            rtb_IP_boBatt1_Actia_Availability := TRUE;
        ELSE 
            rtb_UnitDelay5 := 0;
            (* Switch: '<S675>/Switch2' incorporates:
             *  Constant: '<S261>/Constant1'
             *  Constant: '<S675>/Constant2' *)
            rtb_IP_boBatt1_Actia_Availability := FALSE;
        END_IF;

        (* End of Switch: '<S261>/Switch' *)
        (* End of Outputs for SubSystem: '<Root>/ChiefMaster' *)
        i0_Chartbatt2(ssMethodType := SS_OUTPUT, BattAvailable_LiBa := rtb_S_in, BattAvailable_Actia := rtb_IP_boBatt1_Actia_Availability);
        rtb_BattSelect := i0_Chartbatt2.BattSelect;
        (* Outputs for Atomic SubSystem: '<Root>/ChiefMaster' *)
        (* Sum: '<S269>/Add' incorporates:
         *  ArithShift: '<S268>/Shift Arithmetic'
         *  Constant: '<S267>/Constant'
         *  DataTypeConversion: '<S268>/Data Type Conversion'
         *  Product: '<S269>/Product'
         *  Sum: '<S268>/Add' *)
        rtb_Add_an := DINT_TO_REAL(DWORD_TO_DINT(SHL(DINT_TO_DWORD(USINT_TO_DINT(C_Actia_Batt2_ADS_3[2])), 8)) + USINT_TO_DINT(C_Actia_Batt2_ADS_3[1])) * 0.1;
        (* Sum: '<S578>/Add' incorporates:
         *  ArithShift: '<S577>/Shift Arithmetic'
         *  Constant: '<S573>/Constant'
         *  DataTypeConversion: '<S577>/Data Type Conversion'
         *  Product: '<S578>/Product'
         *  Sum: '<S577>/Add' *)
        rtb_Add_ic := DINT_TO_REAL(DWORD_TO_DINT(SHL(DINT_TO_DWORD(USINT_TO_DINT(C_LB_Batt2_Status02_Msg[7])), 8)) + USINT_TO_DINT(C_LB_Batt2_Status02_Msg[6])) * 0.1;
        (* Switch: '<S578>/Switch' incorporates:
         *  Constant: '<S573>/Constant3'
         *  Constant: '<S573>/Constant4'
         *  RelationalOperator: '<S578>/GreaterThan'
         *  Switch: '<S578>/Switch1' *)

        IF C_LB_Batt2_Status02_Timeout THEN 
            rtb_Add_ic := 0.0;
        ELSIF rtb_Add_ic > 6553.5 THEN 
            (* Switch: '<S578>/Switch1' incorporates:
             *  Constant: '<S573>/Constant4' *)
            rtb_Add_ic := 0.0;
        END_IF;

        (* End of Switch: '<S578>/Switch' *)
        

        (* MultiPortSwitch: '<S713>/Multiport Switch' incorporates:
         *  Constant: '<S713>/Constant' *)

        CASE TRUNC(rtb_BattSelect) OF
            1: 
                (* Switch: '<S269>/Switch' incorporates:
                 *  Constant: '<S267>/Constant3'
                 *  Constant: '<S267>/SafeValue_NA '
                 *  RelationalOperator: '<S269>/GreaterThan'
                 *  Switch: '<S269>/Switch1' *)

                IF C_Actia_Batt2_ADS_3_Timeout THEN 
                    rtb_Add_an := 0.0;
                ELSIF rtb_Add_an > 6553.5 THEN 
                    (* Switch: '<S269>/Switch1' incorporates:
                     *  Constant: '<S267>/SafeValue_Error' *)
                    rtb_Add_an := 0.0;
                END_IF;

                (* End of Switch: '<S269>/Switch' *)
            2: 
                rtb_Add_an := rtb_Add_ic;
            3: 
                rtb_Add_an := 0.0;
            ELSE
                rtb_Add_an := 0.0;
        END_CASE;

        (* End of MultiPortSwitch: '<S713>/Multiport Switch' *)
        

        (* Switch: '<S591>/Switch' incorporates:
         *  Constant: '<S591>/Constant'
         *  Constant: '<S591>/Constant1'
         *  Logic: '<S591>/AND'
         *  Logic: '<S591>/NOT'
         *  Logic: '<S591>/NOT1'
         *  Logic: '<S591>/NOT2'
         *  Logic: '<S591>/NOT3'
         *  Logic: '<S591>/NOT4'
         *  Logic: '<S591>/NOT5'
         *  Logic: '<S591>/NOT6' *)

        IF (((((( NOT C_LB_Batt3_CellVoltage01_Timeout) AND ( NOT C_LB_Batt3_CellVoltage02_Timeout)) AND ( NOT C_LB_Batt3_CellTemperature_Timeout)) AND ( NOT C_LB_Batt3_InsulationMonitor_Timeout)) AND ( NOT C_LB_Batt3_Status01_Timeout)) AND ( NOT C_LB_Batt3_Status02_Timeout)) AND ( NOT C_LB_Batt3_Status03_Timeout) THEN 
            rtb_Switch_b := TRUE;
            (* Switch: '<S675>/Switch5' incorporates:
             *  Constant: '<S591>/Constant'
             *  Constant: '<S675>/Constant11' *)
            rtb_S_in := TRUE;
        ELSE 
            rtb_Switch_b := FALSE;
            (* Switch: '<S675>/Switch5' incorporates:
             *  Constant: '<S591>/Constant1'
             *  Constant: '<S675>/Constant12' *)
            rtb_S_in := FALSE;
        END_IF;

        (* End of Switch: '<S591>/Switch' *)
        

        (* Switch: '<S322>/Switch' incorporates:
         *  Constant: '<S322>/Constant'
         *  Constant: '<S322>/Constant1'
         *  Logic: '<S322>/AND'
         *  Logic: '<S322>/NOT'
         *  Logic: '<S322>/NOT1'
         *  Logic: '<S322>/NOT2'
         *  Logic: '<S322>/NOT3'
         *  Logic: '<S322>/NOT4'
         *  Logic: '<S322>/NOT5' *)

        IF ((((( NOT C_Actia_Batt3_MyStatus_Timeout) AND ( NOT C_Actia_Batt3_Error_Timeout)) AND ( NOT C_Actia_Batt3_ADS_8_Timeout)) AND ( NOT C_Actia_Batt3_ADS_0_Timeout)) AND ( NOT C_Actia_Batt3_ADS_1_Timeout)) AND ( NOT C_Actia_Batt3_ADS_3_Timeout) THEN 
            rtb_Uk1 := 1.0;
            (* Switch: '<S675>/Switch4' incorporates:
             *  Constant: '<S322>/Constant'
             *  Constant: '<S675>/Constant9' *)
            rtb_IP_boBatt1_Actia_Availability := TRUE;
        ELSE 
            rtb_Uk1 := 0.0;
            (* Switch: '<S675>/Switch4' incorporates:
             *  Constant: '<S322>/Constant1'
             *  Constant: '<S675>/Constant10' *)
            rtb_IP_boBatt1_Actia_Availability := FALSE;
        END_IF;

        (* End of Switch: '<S322>/Switch' *)
        (* End of Outputs for SubSystem: '<Root>/ChiefMaster' *)
        i0_ChartBatt3(ssMethodType := SS_OUTPUT, BattAvailable_LiBa := rtb_S_in, BattAvailable_Actia := rtb_IP_boBatt1_Actia_Availability);
        rtb_BattSelect_i := i0_ChartBatt3.BattSelect;
        (* Outputs for Atomic SubSystem: '<Root>/ChiefMaster' *)
        (* Sum: '<S330>/Add' incorporates:
         *  ArithShift: '<S329>/Shift Arithmetic'
         *  Constant: '<S328>/Constant'
         *  DataTypeConversion: '<S329>/Data Type Conversion'
         *  Product: '<S330>/Product'
         *  Sum: '<S329>/Add' *)
        rtb_Add_e := DINT_TO_REAL(DWORD_TO_DINT(SHL(DINT_TO_DWORD(USINT_TO_DINT(C_Actia_Batt3_ADS_3[2])), 8)) + USINT_TO_DINT(C_Actia_Batt3_ADS_3[1])) * 0.1;
        (* Sum: '<S658>/Add' incorporates:
         *  ArithShift: '<S657>/Shift Arithmetic'
         *  Constant: '<S653>/Constant'
         *  DataTypeConversion: '<S657>/Data Type Conversion'
         *  Product: '<S658>/Product'
         *  Sum: '<S657>/Add' *)
        rtb_Add_en := DINT_TO_REAL(DWORD_TO_DINT(SHL(DINT_TO_DWORD(USINT_TO_DINT(C_LB_Batt3_Status02_Msg[7])), 8)) + USINT_TO_DINT(C_LB_Batt3_Status02_Msg[6])) * 0.1;
        (* Switch: '<S658>/Switch' incorporates:
         *  Constant: '<S653>/Constant3'
         *  Constant: '<S653>/Constant4'
         *  RelationalOperator: '<S658>/GreaterThan'
         *  Switch: '<S658>/Switch1' *)

        IF C_LB_Batt3_Status02_Timeout THEN 
            rtb_Add_en := 0.0;
        ELSIF rtb_Add_en > 6553.5 THEN 
            (* Switch: '<S658>/Switch1' incorporates:
             *  Constant: '<S653>/Constant4' *)
            rtb_Add_en := 0.0;
        END_IF;

        (* End of Switch: '<S658>/Switch' *)
        

        (* MultiPortSwitch: '<S714>/Multiport Switch' incorporates:
         *  Constant: '<S714>/Constant' *)

        CASE TRUNC(rtb_BattSelect_i) OF
            1: 
                (* Switch: '<S330>/Switch' incorporates:
                 *  Constant: '<S328>/Constant3'
                 *  Constant: '<S328>/SafeValue_NA '
                 *  RelationalOperator: '<S330>/GreaterThan'
                 *  Switch: '<S330>/Switch1' *)

                IF C_Actia_Batt3_ADS_3_Timeout THEN 
                    rtb_Add_e := 0.0;
                ELSIF rtb_Add_e > 6553.5 THEN 
                    (* Switch: '<S330>/Switch1' incorporates:
                     *  Constant: '<S328>/SafeValue_Error' *)
                    rtb_Add_e := 0.0;
                END_IF;

                (* End of Switch: '<S330>/Switch' *)
            2: 
                rtb_Add_e := rtb_Add_en;
            3: 
                rtb_Add_e := 0.0;
            ELSE
                rtb_Add_e := 0.0;
        END_CASE;

        (* End of MultiPortSwitch: '<S714>/Multiport Switch' *)
        

        (* Outputs for Enabled SubSystem: '<S201>/Subsystem' incorporates:
         *  EnablePort: '<S209>/Timeout' *)
        (* Logic: '<S201>/NOT' *)

        IF  NOT C_Actia_Batt1_MyStatus_Timeout THEN 

            IF  NOT Subsystem_MODE_dz THEN 
                Subsystem_MODE_dz := TRUE;
            END_IF;

            (* DataTypeConversion: '<S209>/Data Type Conversion2' incorporates:
             *  DataTypeConversion: '<S213>/Extract Desired Bits' *)
            IP_boBatt1_HV_REL_ON := DWORD_TO_UDINT(UDINT_TO_DWORD(USINT_TO_UDINT(C_Actia_Batt1_MyStatus[0])) AND 1) <> 0;
            (* DataTypeConversion: '<S209>/Data Type Conversion5' incorporates:
             *  DataTypeConversion: '<S216>/Extract Desired Bits' *)
            IP_boBatt1_SDERR_activ := DWORD_TO_UDINT(UDINT_TO_DWORD(DINT_TO_UDINT(DWORD_TO_DINT(SHR(DINT_TO_DWORD(USINT_TO_DINT(C_Actia_Batt1_MyStatus[0])), 3)))) AND 1) <> 0;
            (* DataTypeConversion: '<S209>/Data Type Conversion6' incorporates:
             *  DataTypeConversion: '<S217>/Extract Desired Bits' *)
            IP_boBatt1_ERROR_activ := DWORD_TO_UDINT(UDINT_TO_DWORD(DINT_TO_UDINT(DWORD_TO_DINT(SHR(DINT_TO_DWORD(USINT_TO_DINT(C_Actia_Batt1_MyStatus[0])), 4)))) AND 1) <> 0;
            (* DataTypeConversion: '<S209>/Data Type Conversion7' incorporates:
             *  DataTypeConversion: '<S218>/Extract Desired Bits' *)
            IP_boBatt1_WARNING_activ := DWORD_TO_UDINT(UDINT_TO_DWORD(DINT_TO_UDINT(DWORD_TO_DINT(SHR(DINT_TO_DWORD(USINT_TO_DINT(C_Actia_Batt1_MyStatus[0])), 5)))) AND 1) <> 0;
            (* DataTypeConversion: '<S209>/Data Type Conversion8' incorporates:
             *  DataTypeConversion: '<S219>/Extract Desired Bits' *)
            IP_boBatt1_Insulation_ready_and_OK := DWORD_TO_UDINT(UDINT_TO_DWORD(DINT_TO_UDINT(DWORD_TO_DINT(SHR(DINT_TO_DWORD(USINT_TO_DINT(C_Actia_Batt1_MyStatus[0])), 6)))) AND 1) <> 0;
        ELSIF Subsystem_MODE_dz THEN 
            (* Disable for DataTypeConversion: '<S209>/Data Type Conversion2' incorporates:
             *  Outport: '<S209>/Batt1_MyStatus1_Databus' *)
            IP_boBatt1_HV_REL_ON := FALSE;
            (* Disable for DataTypeConversion: '<S209>/Data Type Conversion5' incorporates:
             *  Outport: '<S209>/Batt1_MyStatus1_Databus' *)
            IP_boBatt1_SDERR_activ := FALSE;
            (* Disable for DataTypeConversion: '<S209>/Data Type Conversion6' incorporates:
             *  Outport: '<S209>/Batt1_MyStatus1_Databus' *)
            IP_boBatt1_ERROR_activ := FALSE;
            (* Disable for DataTypeConversion: '<S209>/Data Type Conversion7' incorporates:
             *  Outport: '<S209>/Batt1_MyStatus1_Databus' *)
            IP_boBatt1_WARNING_activ := FALSE;
            (* Disable for DataTypeConversion: '<S209>/Data Type Conversion8' incorporates:
             *  Outport: '<S209>/Batt1_MyStatus1_Databus' *)
            IP_boBatt1_Insulation_ready_and_OK := FALSE;
            Subsystem_MODE_dz := FALSE;
        END_IF;

        (* End of Logic: '<S201>/NOT' *)
        (* End of Outputs for SubSystem: '<S201>/Subsystem' *)
        

        (* Logic: '<S428>/NOT1' incorporates:
         *  DataTypeConversion: '<S472>/Extract Desired Bits' *)
        i0_Lib_InputProcessing_state(ssMethodType := SS_OUTPUT, Timeout :=  NOT C_LB_Batt1_Status01_Timeout, Data_In := DINT_TO_USINT(DWORD_TO_DINT(DINT_TO_DWORD(USINT_TO_DINT(C_LB_Batt1_Status01_Msg[0])) AND 15)));
        DataTypeConversion_c := i0_Lib_InputProcessing_state.u8Data_Out;
        (* MultiPortSwitch: '<S715>/Multiport Switch' incorporates:
         *  Constant: '<S715>/Constant'
         *  Constant: '<S718>/Constant'
         *  RelationalOperator: '<S718>/Compare' *)

        CASE TRUNC(rtb_BattSelect_f) OF
            1: 
                rtb_IP_boBMS_SDError_BB1 := IP_boBatt1_SDERR_activ;
            2: 
                rtb_IP_boBMS_SDError_BB1 := DataTypeConversion_c = 4;
            3: 
                rtb_IP_boBMS_SDError_BB1 := FALSE;
            ELSE
                rtb_IP_boBMS_SDError_BB1 := FALSE;
        END_CASE;

        (* End of MultiPortSwitch: '<S715>/Multiport Switch' *)
        

        (* Outputs for Enabled SubSystem: '<S262>/Subsystem' incorporates:
         *  EnablePort: '<S270>/Timeout' *)
        (* Logic: '<S262>/NOT' *)

        IF  NOT C_Actia_Batt2_MyStatus_Timeout THEN 

            IF  NOT Subsystem_MODE_d THEN 
                Subsystem_MODE_d := TRUE;
            END_IF;

            (* DataTypeConversion: '<S270>/Data Type Conversion2' incorporates:
             *  DataTypeConversion: '<S274>/Extract Desired Bits' *)
            IP_boBatt2_HV_REL_ON := DWORD_TO_UDINT(UDINT_TO_DWORD(USINT_TO_UDINT(C_Actia_Batt2_MyStatus[0])) AND 1) <> 0;
            (* DataTypeConversion: '<S270>/Data Type Conversion5' incorporates:
             *  DataTypeConversion: '<S277>/Extract Desired Bits' *)
            IP_boBatt2_SDERR_activ := DWORD_TO_UDINT(UDINT_TO_DWORD(DINT_TO_UDINT(DWORD_TO_DINT(SHR(DINT_TO_DWORD(USINT_TO_DINT(C_Actia_Batt2_MyStatus[0])), 3)))) AND 1) <> 0;
            (* DataTypeConversion: '<S270>/Data Type Conversion6' incorporates:
             *  DataTypeConversion: '<S278>/Extract Desired Bits' *)
            IP_boBatt2_ERROR_activ := DWORD_TO_UDINT(UDINT_TO_DWORD(DINT_TO_UDINT(DWORD_TO_DINT(SHR(DINT_TO_DWORD(USINT_TO_DINT(C_Actia_Batt2_MyStatus[0])), 4)))) AND 1) <> 0;
            (* DataTypeConversion: '<S270>/Data Type Conversion7' incorporates:
             *  DataTypeConversion: '<S279>/Extract Desired Bits' *)
            IP_boBatt2_WARNING_activ := DWORD_TO_UDINT(UDINT_TO_DWORD(DINT_TO_UDINT(DWORD_TO_DINT(SHR(DINT_TO_DWORD(USINT_TO_DINT(C_Actia_Batt2_MyStatus[0])), 5)))) AND 1) <> 0;
            (* DataTypeConversion: '<S270>/Data Type Conversion8' incorporates:
             *  DataTypeConversion: '<S280>/Extract Desired Bits' *)
            IP_boBatt2_Insulation_ready_and_OK := DWORD_TO_UDINT(UDINT_TO_DWORD(DINT_TO_UDINT(DWORD_TO_DINT(SHR(DINT_TO_DWORD(USINT_TO_DINT(C_Actia_Batt2_MyStatus[0])), 6)))) AND 1) <> 0;
        ELSIF Subsystem_MODE_d THEN 
            (* Disable for DataTypeConversion: '<S270>/Data Type Conversion2' incorporates:
             *  Outport: '<S270>/Batt2_MyStatus1_Databus' *)
            IP_boBatt2_HV_REL_ON := FALSE;
            (* Disable for DataTypeConversion: '<S270>/Data Type Conversion5' incorporates:
             *  Outport: '<S270>/Batt2_MyStatus1_Databus' *)
            IP_boBatt2_SDERR_activ := FALSE;
            (* Disable for DataTypeConversion: '<S270>/Data Type Conversion6' incorporates:
             *  Outport: '<S270>/Batt2_MyStatus1_Databus' *)
            IP_boBatt2_ERROR_activ := FALSE;
            (* Disable for DataTypeConversion: '<S270>/Data Type Conversion7' incorporates:
             *  Outport: '<S270>/Batt2_MyStatus1_Databus' *)
            IP_boBatt2_WARNING_activ := FALSE;
            (* Disable for DataTypeConversion: '<S270>/Data Type Conversion8' incorporates:
             *  Outport: '<S270>/Batt2_MyStatus1_Databus' *)
            IP_boBatt2_Insulation_ready_and_OK := FALSE;
            Subsystem_MODE_d := FALSE;
        END_IF;

        (* End of Logic: '<S262>/NOT' *)
        (* End of Outputs for SubSystem: '<S262>/Subsystem' *)
        

        (* Logic: '<S508>/NOT1' incorporates:
         *  DataTypeConversion: '<S552>/Extract Desired Bits' *)
        i1_Lib_InputProcessing_state(ssMethodType := SS_OUTPUT, Timeout :=  NOT C_LB_Batt2_Status01_Timeout, Data_In := DINT_TO_USINT(DWORD_TO_DINT(DINT_TO_DWORD(USINT_TO_DINT(C_LB_Batt2_Status01_Msg[0])) AND 15)));
        DataTypeConversion_i := i1_Lib_InputProcessing_state.u8Data_Out;
        (* MultiPortSwitch: '<S716>/Multiport Switch' incorporates:
         *  Constant: '<S716>/Constant'
         *  Constant: '<S719>/Constant'
         *  RelationalOperator: '<S719>/Compare' *)

        CASE TRUNC(rtb_BattSelect) OF
            1: 
                rtb_IP_boBMS_SDError_BB2 := IP_boBatt2_SDERR_activ;
            2: 
                rtb_IP_boBMS_SDError_BB2 := DataTypeConversion_i = 4;
            3: 
                rtb_IP_boBMS_SDError_BB2 := FALSE;
            ELSE
                rtb_IP_boBMS_SDError_BB2 := FALSE;
        END_CASE;

        (* End of MultiPortSwitch: '<S716>/Multiport Switch' *)
        

        (* Outputs for Enabled SubSystem: '<S323>/Subsystem' incorporates:
         *  EnablePort: '<S331>/Timeout' *)
        (* Logic: '<S323>/NOT' *)

        IF  NOT C_Actia_Batt3_MyStatus_Timeout THEN 

            IF  NOT Subsystem_MODE_e THEN 
                Subsystem_MODE_e := TRUE;
            END_IF;

            (* DataTypeConversion: '<S331>/Data Type Conversion2' incorporates:
             *  DataTypeConversion: '<S335>/Extract Desired Bits' *)
            IP_boBatt3_HV_REL_ON := DWORD_TO_UDINT(UDINT_TO_DWORD(USINT_TO_UDINT(C_Actia_Batt3_MyStatus[0])) AND 1) <> 0;
            (* DataTypeConversion: '<S331>/Data Type Conversion5' incorporates:
             *  DataTypeConversion: '<S338>/Extract Desired Bits' *)
            IP_boBatt3_SDERR_activ := DWORD_TO_UDINT(UDINT_TO_DWORD(DINT_TO_UDINT(DWORD_TO_DINT(SHR(DINT_TO_DWORD(USINT_TO_DINT(C_Actia_Batt3_MyStatus[0])), 3)))) AND 1) <> 0;
            (* DataTypeConversion: '<S331>/Data Type Conversion6' incorporates:
             *  DataTypeConversion: '<S339>/Extract Desired Bits' *)
            IP_boBatt3_ERROR_activ := DWORD_TO_UDINT(UDINT_TO_DWORD(DINT_TO_UDINT(DWORD_TO_DINT(SHR(DINT_TO_DWORD(USINT_TO_DINT(C_Actia_Batt3_MyStatus[0])), 4)))) AND 1) <> 0;
            (* DataTypeConversion: '<S331>/Data Type Conversion7' incorporates:
             *  DataTypeConversion: '<S340>/Extract Desired Bits' *)
            IP_boBatt3_WARNING_activ := DWORD_TO_UDINT(UDINT_TO_DWORD(DINT_TO_UDINT(DWORD_TO_DINT(SHR(DINT_TO_DWORD(USINT_TO_DINT(C_Actia_Batt3_MyStatus[0])), 5)))) AND 1) <> 0;
            (* DataTypeConversion: '<S331>/Data Type Conversion8' incorporates:
             *  DataTypeConversion: '<S341>/Extract Desired Bits' *)
            IP_boBatt3_Insulation_ready_and_OK := DWORD_TO_UDINT(UDINT_TO_DWORD(DINT_TO_UDINT(DWORD_TO_DINT(SHR(DINT_TO_DWORD(USINT_TO_DINT(C_Actia_Batt3_MyStatus[0])), 6)))) AND 1) <> 0;
        ELSIF Subsystem_MODE_e THEN 
            (* Disable for DataTypeConversion: '<S331>/Data Type Conversion2' incorporates:
             *  Outport: '<S331>/Batt3_MyStatus1_Databus' *)
            IP_boBatt3_HV_REL_ON := FALSE;
            (* Disable for DataTypeConversion: '<S331>/Data Type Conversion5' incorporates:
             *  Outport: '<S331>/Batt3_MyStatus1_Databus' *)
            IP_boBatt3_SDERR_activ := FALSE;
            (* Disable for DataTypeConversion: '<S331>/Data Type Conversion6' incorporates:
             *  Outport: '<S331>/Batt3_MyStatus1_Databus' *)
            IP_boBatt3_ERROR_activ := FALSE;
            (* Disable for DataTypeConversion: '<S331>/Data Type Conversion7' incorporates:
             *  Outport: '<S331>/Batt3_MyStatus1_Databus' *)
            IP_boBatt3_WARNING_activ := FALSE;
            (* Disable for DataTypeConversion: '<S331>/Data Type Conversion8' incorporates:
             *  Outport: '<S331>/Batt3_MyStatus1_Databus' *)
            IP_boBatt3_Insulation_ready_and_OK := FALSE;
            Subsystem_MODE_e := FALSE;
        END_IF;

        (* End of Logic: '<S323>/NOT' *)
        (* End of Outputs for SubSystem: '<S323>/Subsystem' *)
        

        (* Logic: '<S588>/NOT1' incorporates:
         *  DataTypeConversion: '<S632>/Extract Desired Bits' *)
        i2_Lib_InputProcessing_state(ssMethodType := SS_OUTPUT, Timeout :=  NOT C_LB_Batt3_Status01_Timeout, Data_In := DINT_TO_USINT(DWORD_TO_DINT(DINT_TO_DWORD(USINT_TO_DINT(C_LB_Batt3_Status01_Msg[0])) AND 15)));
        DataTypeConversion := i2_Lib_InputProcessing_state.u8Data_Out;
        (* MultiPortSwitch: '<S717>/Multiport Switch' incorporates:
         *  Constant: '<S717>/Constant'
         *  Constant: '<S720>/Constant'
         *  RelationalOperator: '<S720>/Compare' *)

        CASE TRUNC(rtb_BattSelect_i) OF
            1: 
                rtb_IP_boBMS_SDError_BB3 := IP_boBatt3_SDERR_activ;
            2: 
                rtb_IP_boBMS_SDError_BB3 := DataTypeConversion = 4;
            3: 
                rtb_IP_boBMS_SDError_BB3 := FALSE;
            ELSE
                rtb_IP_boBMS_SDError_BB3 := FALSE;
        END_CASE;

        (* End of MultiPortSwitch: '<S717>/Multiport Switch' *)
        

        (* Sum: '<S486>/Add' incorporates:
         *  Product: '<S486>/Product' *)
        rtb_Add_nm := USINT_TO_REAL(C_LB_Batt1_Status01_Msg[1]);
        (* Switch: '<S486>/Switch' incorporates:
         *  Constant: '<S482>/Constant4' *)

        IF C_LB_Batt1_Status01_Timeout THEN 
            rtb_Add_nm := 0.0;
        END_IF;

        (* End of Switch: '<S486>/Switch' *)
        

        (* MultiPortSwitch: '<S745>/Multiport Switch' incorporates:
         *  Constant: '<S745>/Constant'
         *  Constant: '<S748>/Constant'
         *  Constant: '<S749>/Constant'
         *  Logic: '<S745>/OR'
         *  RelationalOperator: '<S748>/Compare'
         *  RelationalOperator: '<S749>/Compare' *)

        CASE TRUNC(rtb_BattSelect_f) OF
            1: 
                rtb_IP_boBMS_HV_REL_ON_BB1 := IP_boBatt1_HV_REL_ON;
            2: 
                rtb_IP_boBMS_HV_REL_ON_BB1 := (rtb_Add_nm = 192.0) OR (rtb_Add_nm = 224.0);
            3: 
                rtb_IP_boBMS_HV_REL_ON_BB1 := FALSE;
            ELSE
                rtb_IP_boBMS_HV_REL_ON_BB1 := FALSE;
        END_CASE;

        (* End of MultiPortSwitch: '<S745>/Multiport Switch' *)
        

        (* Sum: '<S566>/Add' incorporates:
         *  Product: '<S566>/Product' *)
        rtb_Add_d4 := USINT_TO_REAL(C_LB_Batt2_Status01_Msg[1]);
        (* Switch: '<S566>/Switch' incorporates:
         *  Constant: '<S562>/Constant4' *)

        IF C_LB_Batt2_Status01_Timeout THEN 
            rtb_Add_d4 := 0.0;
        END_IF;

        (* End of Switch: '<S566>/Switch' *)
        

        (* MultiPortSwitch: '<S746>/Multiport Switch' incorporates:
         *  Constant: '<S746>/Constant'
         *  Constant: '<S750>/Constant'
         *  Constant: '<S751>/Constant'
         *  Logic: '<S746>/OR'
         *  RelationalOperator: '<S750>/Compare'
         *  RelationalOperator: '<S751>/Compare' *)

        CASE TRUNC(rtb_BattSelect) OF
            1: 
                rtb_IP_boBMS_HV_REL_ON_BB2 := IP_boBatt2_HV_REL_ON;
            2: 
                rtb_IP_boBMS_HV_REL_ON_BB2 := (rtb_Add_d4 = 192.0) OR (rtb_Add_d4 = 224.0);
            3: 
                rtb_IP_boBMS_HV_REL_ON_BB2 := FALSE;
            ELSE
                rtb_IP_boBMS_HV_REL_ON_BB2 := FALSE;
        END_CASE;

        (* End of MultiPortSwitch: '<S746>/Multiport Switch' *)
        

        (* Sum: '<S646>/Add' incorporates:
         *  Product: '<S646>/Product' *)
        rtb_Add_cw := USINT_TO_REAL(C_LB_Batt3_Status01_Msg[1]);
        (* Switch: '<S646>/Switch' incorporates:
         *  Constant: '<S642>/Constant4' *)

        IF C_LB_Batt3_Status01_Timeout THEN 
            rtb_Add_cw := 0.0;
        END_IF;

        (* End of Switch: '<S646>/Switch' *)
        

        (* MultiPortSwitch: '<S747>/Multiport Switch' incorporates:
         *  Constant: '<S747>/Constant'
         *  Constant: '<S752>/Constant'
         *  Constant: '<S753>/Constant'
         *  Logic: '<S747>/OR'
         *  RelationalOperator: '<S752>/Compare'
         *  RelationalOperator: '<S753>/Compare' *)

        CASE TRUNC(rtb_BattSelect_i) OF
            1: 
                rtb_IP_boBMS_HV_REL_ON_BB3 := IP_boBatt3_HV_REL_ON;
            2: 
                rtb_IP_boBMS_HV_REL_ON_BB3 := (rtb_Add_cw = 192.0) OR (rtb_Add_cw = 224.0);
            3: 
                rtb_IP_boBMS_HV_REL_ON_BB3 := FALSE;
            ELSE
                rtb_IP_boBMS_HV_REL_ON_BB3 := FALSE;
        END_CASE;

        (* End of MultiPortSwitch: '<S747>/Multiport Switch' *)
        

        (* Sum: '<S250>/Add' incorporates:
         *  ArithShift: '<S249>/Shift Arithmetic'
         *  Constant: '<S245>/Constant'
         *  DataTypeConversion: '<S249>/Data Type Conversion'
         *  Product: '<S250>/Product'
         *  Sum: '<S249>/Add' *)
        rtb_Add_ki5 := INT_TO_REAL(DINT_TO_INT(INT_TO_DINT(WORD_TO_INT(SHL(INT_TO_WORD(USINT_TO_INT(C_Actia_Batt1_ADS_8[4])), 8))) + USINT_TO_DINT(C_Actia_Batt1_ADS_8[3]))) * 0.1;
        (* Sum: '<S496>/Add' incorporates:
         *  ArithShift: '<S495>/Shift Arithmetic'
         *  ArithShift: '<S495>/Shift Arithmetic1'
         *  ArithShift: '<S495>/Shift Arithmetic2'
         *  Constant: '<S492>/Constant'
         *  DataTypeConversion: '<S492>/Data Type Conversion'
         *  DataTypeConversion: '<S495>/Data Type Conversion'
         *  DataTypeConversion: '<S495>/Data Type Conversion1'
         *  DataTypeConversion: '<S495>/Data Type Conversion2'
         *  Product: '<S496>/Product'
         *  Sum: '<S495>/Add' *)
        rtb_Add_ir := DINT_TO_REAL(UDINT_TO_DINT(((DWORD_TO_UDINT(SHL(UDINT_TO_DWORD(USINT_TO_UDINT(C_LB_BMS_Status02_Msg[5])), 24)) + DWORD_TO_UDINT(SHL(UDINT_TO_DWORD(USINT_TO_UDINT(C_LB_BMS_Status02_Msg[4])), 16))) + DWORD_TO_UDINT(SHL(UDINT_TO_DWORD(USINT_TO_UDINT(C_LB_BMS_Status02_Msg[3])), 8))) + USINT_TO_UDINT(C_LB_BMS_Status02_Msg[2]))) * 0.01;
        (* MultiPortSwitch: '<S763>/Multiport Switch' incorporates:
         *  Constant: '<S763>/Constant'
         *  Gain: '<S763>/mAtoA' *)

        CASE TRUNC(rtb_BattSelect_f) OF
            1: 
                (* Switch: '<S250>/Switch' incorporates:
                 *  Constant: '<S245>/SafeValue_NA ' *)

                IF C_Actia_Batt1_ADS_8_Timeout THEN 
                    rtb_Add_ki5 := 0.0;
                END_IF;

                (* End of Switch: '<S250>/Switch' *)
            2: 
                (* Switch: '<S496>/Switch' incorporates:
                 *  Constant: '<S492>/Constant4' *)

                IF C_LB_Batt1_Status02_Timeout THEN 
                    rtb_Add_ir := 0.0;
                END_IF;

                (* End of Switch: '<S496>/Switch' *)
                rtb_Add_ki5 := 0.001 * rtb_Add_ir;
            3: 
                rtb_Add_ki5 := 0.0;
            ELSE
                rtb_Add_ki5 := 0.0;
        END_CASE;

        (* End of MultiPortSwitch: '<S763>/Multiport Switch' *)
        

        (* Sum: '<S311>/Add' incorporates:
         *  ArithShift: '<S310>/Shift Arithmetic'
         *  Constant: '<S306>/Constant'
         *  DataTypeConversion: '<S310>/Data Type Conversion'
         *  Product: '<S311>/Product'
         *  Sum: '<S310>/Add' *)
        rtb_Add_ir := INT_TO_REAL(DINT_TO_INT(INT_TO_DINT(WORD_TO_INT(SHL(INT_TO_WORD(USINT_TO_INT(C_Actia_Batt2_ADS_8[4])), 8))) + USINT_TO_DINT(C_Actia_Batt2_ADS_8[3]))) * 0.1;
        (* Sum: '<S576>/Add' incorporates:
         *  ArithShift: '<S575>/Shift Arithmetic'
         *  ArithShift: '<S575>/Shift Arithmetic1'
         *  ArithShift: '<S575>/Shift Arithmetic2'
         *  Constant: '<S572>/Constant'
         *  DataTypeConversion: '<S572>/Data Type Conversion'
         *  DataTypeConversion: '<S575>/Data Type Conversion'
         *  DataTypeConversion: '<S575>/Data Type Conversion1'
         *  DataTypeConversion: '<S575>/Data Type Conversion2'
         *  Product: '<S576>/Product'
         *  Sum: '<S575>/Add' *)
        rtb_Add_m := DINT_TO_REAL(UDINT_TO_DINT(((DWORD_TO_UDINT(SHL(UDINT_TO_DWORD(USINT_TO_UDINT(C_LB_Batt2_Status02_Msg[5])), 24)) + DWORD_TO_UDINT(SHL(UDINT_TO_DWORD(USINT_TO_UDINT(C_LB_Batt2_Status02_Msg[4])), 16))) + DWORD_TO_UDINT(SHL(UDINT_TO_DWORD(USINT_TO_UDINT(C_LB_Batt2_Status02_Msg[3])), 8))) + USINT_TO_UDINT(C_LB_Batt2_Status02_Msg[2]))) * 0.01;
        (* MultiPortSwitch: '<S764>/Multiport Switch' incorporates:
         *  Constant: '<S764>/Constant'
         *  Gain: '<S764>/mAtoA' *)

        CASE TRUNC(rtb_BattSelect) OF
            1: 
                (* Switch: '<S311>/Switch' incorporates:
                 *  Constant: '<S306>/SafeValue_NA ' *)

                IF C_Actia_Batt2_ADS_8_Timeout THEN 
                    rtb_Add_ir := 0.0;
                END_IF;

                (* End of Switch: '<S311>/Switch' *)
            2: 
                (* Switch: '<S576>/Switch' incorporates:
                 *  Constant: '<S572>/Constant4' *)

                IF C_LB_Batt2_Status02_Timeout THEN 
                    rtb_Add_m := 0.0;
                END_IF;

                (* End of Switch: '<S576>/Switch' *)
                rtb_Add_ir := 0.001 * rtb_Add_m;
            3: 
                rtb_Add_ir := 0.0;
            ELSE
                rtb_Add_ir := 0.0;
        END_CASE;

        (* End of MultiPortSwitch: '<S764>/Multiport Switch' *)
        

        (* Sum: '<S372>/Add' incorporates:
         *  ArithShift: '<S371>/Shift Arithmetic'
         *  Constant: '<S367>/Constant'
         *  DataTypeConversion: '<S371>/Data Type Conversion'
         *  Product: '<S372>/Product'
         *  Sum: '<S371>/Add' *)
        rtb_Add_m := INT_TO_REAL(DINT_TO_INT(INT_TO_DINT(WORD_TO_INT(SHL(INT_TO_WORD(USINT_TO_INT(C_Actia_Batt3_ADS_8[4])), 8))) + USINT_TO_DINT(C_Actia_Batt3_ADS_8[3]))) * 0.1;
        (* Sum: '<S656>/Add' incorporates:
         *  ArithShift: '<S655>/Shift Arithmetic'
         *  ArithShift: '<S655>/Shift Arithmetic1'
         *  ArithShift: '<S655>/Shift Arithmetic2'
         *  Constant: '<S652>/Constant'
         *  DataTypeConversion: '<S652>/Data Type Conversion'
         *  DataTypeConversion: '<S655>/Data Type Conversion'
         *  DataTypeConversion: '<S655>/Data Type Conversion1'
         *  DataTypeConversion: '<S655>/Data Type Conversion2'
         *  Product: '<S656>/Product'
         *  Sum: '<S655>/Add' *)
        rtb_Add_b := DINT_TO_REAL(UDINT_TO_DINT(((DWORD_TO_UDINT(SHL(UDINT_TO_DWORD(USINT_TO_UDINT(C_LB_Batt3_Status02_Msg[5])), 24)) + DWORD_TO_UDINT(SHL(UDINT_TO_DWORD(USINT_TO_UDINT(C_LB_Batt3_Status02_Msg[4])), 16))) + DWORD_TO_UDINT(SHL(UDINT_TO_DWORD(USINT_TO_UDINT(C_LB_Batt3_Status02_Msg[3])), 8))) + USINT_TO_UDINT(C_LB_Batt3_Status02_Msg[2]))) * 0.01;
        (* MultiPortSwitch: '<S765>/Multiport Switch' incorporates:
         *  Constant: '<S765>/Constant'
         *  Gain: '<S765>/mAtoA' *)

        CASE TRUNC(rtb_BattSelect_i) OF
            1: 
                (* Switch: '<S372>/Switch' incorporates:
                 *  Constant: '<S367>/SafeValue_NA ' *)

                IF C_Actia_Batt3_ADS_8_Timeout THEN 
                    rtb_Add_m := 0.0;
                END_IF;

                (* End of Switch: '<S372>/Switch' *)
            2: 
                (* Switch: '<S656>/Switch' incorporates:
                 *  Constant: '<S652>/Constant4' *)

                IF C_LB_Batt3_Status02_Timeout THEN 
                    rtb_Add_b := 0.0;
                END_IF;

                (* End of Switch: '<S656>/Switch' *)
                rtb_Add_m := 0.001 * rtb_Add_b;
            3: 
                rtb_Add_m := 0.0;
            ELSE
                rtb_Add_m := 0.0;
        END_CASE;

        (* End of MultiPortSwitch: '<S765>/Multiport Switch' *)
        

        (* Sum: '<S248>/Add' incorporates:
         *  Product: '<S248>/Product' *)
        rtb_Add_ci := USINT_TO_REAL(C_Actia_Batt1_ADS_8[6]);
        (* MultiPortSwitch: '<S754>/Multiport Switch' incorporates:
         *  Constant: '<S754>/Constant' *)

        CASE TRUNC(rtb_BattSelect_f) OF
            1: 
                (* Switch: '<S248>/Switch' incorporates:
                 *  Constant: '<S244>/Constant3'
                 *  Constant: '<S244>/SafeValue_NA '
                 *  Product: '<S248>/Product'
                 *  RelationalOperator: '<S248>/GreaterThan'
                 *  Switch: '<S248>/Switch1' *)

                IF C_Actia_Batt1_ADS_8_Timeout THEN 
                    rtb_Add_ci := 0.0;
                ELSIF USINT_TO_REAL(C_Actia_Batt1_ADS_8[6]) > 100.0 THEN 
                    (* Switch: '<S248>/Switch1' incorporates:
                     *  Constant: '<S244>/SafeValue_Error' *)
                    rtb_Add_ci := 0.0;
                END_IF;

                (* End of Switch: '<S248>/Switch' *)
            2: 
                (* Switch: '<S500>/Switch' incorporates:
                 *  Constant: '<S494>/Constant4' *)

                IF C_LB_Batt1_Status02_Timeout THEN 
                    rtb_Add_ci := 0.0;
                ELSE 
                    (* Switch: '<S500>/Switch1' incorporates:
                     *  ArithShift: '<S499>/Shift Arithmetic'
                     *  Constant: '<S494>/Constant'
                     *  DataTypeConversion: '<S494>/Data Type Conversion'
                     *  DataTypeConversion: '<S499>/Data Type Conversion'
                     *  Product: '<S500>/Product'
                     *  Sum: '<S499>/Add' *)
                    rtb_Add_ci := INT_TO_REAL(UDINT_TO_INT(DINT_TO_UDINT(DWORD_TO_DINT(SHL(DINT_TO_DWORD(USINT_TO_DINT(C_LB_BMS_Status02_Msg[1])), 8))) + USINT_TO_UDINT(C_LB_BMS_Status02_Msg[0]))) * 0.01;
                END_IF;

                (* End of Switch: '<S500>/Switch' *)
            3: 
                rtb_Add_ci := 0.0;
            ELSE
                rtb_Add_ci := 0.0;
        END_CASE;

        (* End of MultiPortSwitch: '<S754>/Multiport Switch' *)
        

        (* DataTypeConversion: '<S691>/Data Type Conversion' *)
        rtb_DataTypeConversion_k := DINT_TO_USINT(TRUNC(rtb_Add_ci));
        (* Sum: '<S309>/Add' incorporates:
         *  Product: '<S309>/Product' *)
        rtb_Add_ci := USINT_TO_REAL(C_Actia_Batt2_ADS_8[6]);
        (* MultiPortSwitch: '<S755>/Multiport Switch' incorporates:
         *  Constant: '<S755>/Constant' *)

        CASE TRUNC(rtb_BattSelect) OF
            1: 
                (* Switch: '<S309>/Switch' incorporates:
                 *  Constant: '<S305>/Constant3'
                 *  Constant: '<S305>/SafeValue_NA '
                 *  Product: '<S309>/Product'
                 *  RelationalOperator: '<S309>/GreaterThan'
                 *  Switch: '<S309>/Switch1' *)

                IF C_Actia_Batt2_ADS_8_Timeout THEN 
                    rtb_Add_ci := 0.0;
                ELSIF USINT_TO_REAL(C_Actia_Batt2_ADS_8[6]) > 100.0 THEN 
                    (* Switch: '<S309>/Switch1' incorporates:
                     *  Constant: '<S305>/SafeValue_Error' *)
                    rtb_Add_ci := 0.0;
                END_IF;

                (* End of Switch: '<S309>/Switch' *)
            2: 
                (* Switch: '<S580>/Switch' incorporates:
                 *  Constant: '<S574>/Constant4' *)

                IF C_LB_Batt2_Status02_Timeout THEN 
                    rtb_Add_ci := 0.0;
                ELSE 
                    (* Switch: '<S580>/Switch1' incorporates:
                     *  ArithShift: '<S579>/Shift Arithmetic'
                     *  Constant: '<S574>/Constant'
                     *  DataTypeConversion: '<S574>/Data Type Conversion'
                     *  DataTypeConversion: '<S579>/Data Type Conversion'
                     *  Product: '<S580>/Product'
                     *  Sum: '<S579>/Add' *)
                    rtb_Add_ci := INT_TO_REAL(UDINT_TO_INT(DINT_TO_UDINT(DWORD_TO_DINT(SHL(DINT_TO_DWORD(USINT_TO_DINT(C_LB_Batt2_Status02_Msg[1])), 8))) + USINT_TO_UDINT(C_LB_Batt2_Status02_Msg[0]))) * 0.01;
                END_IF;

                (* End of Switch: '<S580>/Switch' *)
            3: 
                rtb_Add_ci := 0.0;
            ELSE
                rtb_Add_ci := 0.0;
        END_CASE;

        (* End of MultiPortSwitch: '<S755>/Multiport Switch' *)
        

        (* DataTypeConversion: '<S691>/Data Type Conversion1' *)
        rtb_DataTypeConversion1 := DINT_TO_USINT(TRUNC(rtb_Add_ci));
        (* Sum: '<S370>/Add' incorporates:
         *  Product: '<S370>/Product' *)
        rtb_Add_ci := USINT_TO_REAL(C_Actia_Batt3_ADS_8[6]);
        (* MultiPortSwitch: '<S756>/Multiport Switch' incorporates:
         *  Constant: '<S756>/Constant' *)

        CASE TRUNC(rtb_BattSelect_i) OF
            1: 
                (* Switch: '<S370>/Switch' incorporates:
                 *  Constant: '<S366>/Constant3'
                 *  Constant: '<S366>/SafeValue_NA '
                 *  Product: '<S370>/Product'
                 *  RelationalOperator: '<S370>/GreaterThan'
                 *  Switch: '<S370>/Switch1' *)

                IF C_Actia_Batt3_ADS_8_Timeout THEN 
                    rtb_Add_ci := 0.0;
                ELSIF USINT_TO_REAL(C_Actia_Batt3_ADS_8[6]) > 100.0 THEN 
                    (* Switch: '<S370>/Switch1' incorporates:
                     *  Constant: '<S366>/SafeValue_Error' *)
                    rtb_Add_ci := 0.0;
                END_IF;

                (* End of Switch: '<S370>/Switch' *)
            2: 
                (* Switch: '<S660>/Switch' incorporates:
                 *  Constant: '<S654>/Constant4' *)

                IF C_LB_Batt3_Status02_Timeout THEN 
                    rtb_Add_ci := 0.0;
                ELSE 
                    (* Switch: '<S660>/Switch1' incorporates:
                     *  ArithShift: '<S659>/Shift Arithmetic'
                     *  Constant: '<S654>/Constant'
                     *  DataTypeConversion: '<S654>/Data Type Conversion'
                     *  DataTypeConversion: '<S659>/Data Type Conversion'
                     *  Product: '<S660>/Product'
                     *  Sum: '<S659>/Add' *)
                    rtb_Add_ci := INT_TO_REAL(UDINT_TO_INT(DINT_TO_UDINT(DWORD_TO_DINT(SHL(DINT_TO_DWORD(USINT_TO_DINT(C_LB_Batt3_Status02_Msg[1])), 8))) + USINT_TO_UDINT(C_LB_Batt3_Status02_Msg[0]))) * 0.01;
                END_IF;

                (* End of Switch: '<S660>/Switch' *)
            3: 
                rtb_Add_ci := 0.0;
            ELSE
                rtb_Add_ci := 0.0;
        END_CASE;

        (* End of MultiPortSwitch: '<S756>/Multiport Switch' *)
        

        (* DataTypeConversion: '<S691>/Data Type Conversion2' *)
        rtb_DataTypeConversion2_h := DINT_TO_USINT(TRUNC(rtb_Add_ci));
        (* Sum: '<S225>/Add' incorporates:
         *  ArithShift: '<S224>/Shift Arithmetic'
         *  Constant: '<S212>/Constant'
         *  DataTypeConversion: '<S224>/Data Type Conversion'
         *  Product: '<S225>/Product'
         *  Sum: '<S224>/Add' *)
        rtb_Add_b := DINT_TO_REAL(DWORD_TO_DINT(SHL(DINT_TO_DWORD(USINT_TO_DINT(C_Actia_Batt1_MyStatus[2])), 8)) + USINT_TO_DINT(C_Actia_Batt1_MyStatus[1])) * 0.1;
        (* Sum: '<S503>/Add' incorporates:
         *  ArithShift: '<S502>/Shift Arithmetic'
         *  Constant: '<S501>/Constant'
         *  DataTypeConversion: '<S502>/Data Type Conversion'
         *  Product: '<S503>/Product'
         *  Sum: '<S502>/Add' *)
        rtb_Add_h := DINT_TO_REAL(DWORD_TO_DINT(SHL(DINT_TO_DWORD(USINT_TO_DINT(C_LB_Batt1_Status03_Msg[1])), 8)) + USINT_TO_DINT(C_LB_Batt1_Status03_Msg[0])) * 0.1;
        (* Sum: '<S489>/Add' incorporates:
         *  ArithShift: '<S488>/Shift Arithmetic'
         *  Constant: '<S484>/Constant'
         *  DataTypeConversion: '<S488>/Data Type Conversion'
         *  Product: '<S489>/Product'
         *  Sum: '<S488>/Add' *)
        rtb_Add_g := DINT_TO_REAL(DWORD_TO_DINT(SHL(DINT_TO_DWORD(USINT_TO_DINT(C_LB_Batt1_Status01_Msg[5])), 8)) + USINT_TO_DINT(C_LB_Batt1_Status01_Msg[4])) * 0.1;
        (* MultiPortSwitch: '<S760>/Multiport Switch' incorporates:
         *  Constant: '<S760>/Constant'
         *  MinMax: '<S760>/Min' *)

        CASE TRUNC(rtb_BattSelect_f) OF
            1: 
                (* Switch: '<S225>/Switch' incorporates:
                 *  Constant: '<S212>/Constant3'
                 *  Constant: '<S212>/SafeValue_NA '
                 *  RelationalOperator: '<S225>/GreaterThan'
                 *  Switch: '<S225>/Switch1' *)

                IF C_Actia_Batt1_MyStatus_Timeout THEN 
                    rtb_Add_b := 0.0;
                ELSIF rtb_Add_b > 6553.5 THEN 
                    (* Switch: '<S225>/Switch1' incorporates:
                     *  Constant: '<S212>/SafeValue_Error' *)
                    rtb_Add_b := 0.0;
                END_IF;

                (* End of Switch: '<S225>/Switch' *)
            2: 
                (* Switch: '<S489>/Switch' incorporates:
                 *  Constant: '<S484>/Constant3'
                 *  Constant: '<S484>/Constant4'
                 *  RelationalOperator: '<S489>/GreaterThan'
                 *  Switch: '<S489>/Switch1' *)

                IF C_LB_Batt1_Status01_Timeout THEN 
                    rtb_Add_g := 0.0;
                ELSIF rtb_Add_g > 6553.5 THEN 
                    (* Switch: '<S489>/Switch1' incorporates:
                     *  Constant: '<S484>/Constant4' *)
                    rtb_Add_g := 0.0;
                END_IF;

                (* End of Switch: '<S489>/Switch' *)
                

                (* Switch: '<S503>/Switch' incorporates:
                 *  Constant: '<S501>/Constant3'
                 *  Constant: '<S501>/Constant4'
                 *  RelationalOperator: '<S503>/GreaterThan'
                 *  Switch: '<S503>/Switch1' *)

                IF C_LB_Batt1_Status03_Timeout THEN 
                    rtb_Add_h := 0.0;
                ELSIF rtb_Add_h > 6553.5 THEN 
                    (* Switch: '<S503>/Switch1' incorporates:
                     *  Constant: '<S501>/Constant4' *)
                    rtb_Add_h := 0.0;
                END_IF;

                (* End of Switch: '<S503>/Switch' *)
                rtb_Add_b := MIN(rtb_Add_h, rtb_Add_g);
            3: 
                rtb_Add_b := 0.0;
            ELSE
                rtb_Add_b := 0.0;
        END_CASE;

        (* End of MultiPortSwitch: '<S760>/Multiport Switch' *)
        

        (* Sum: '<S286>/Add' incorporates:
         *  ArithShift: '<S285>/Shift Arithmetic'
         *  Constant: '<S273>/Constant'
         *  DataTypeConversion: '<S285>/Data Type Conversion'
         *  Product: '<S286>/Product'
         *  Sum: '<S285>/Add' *)
        rtb_Add_h := DINT_TO_REAL(DWORD_TO_DINT(SHL(DINT_TO_DWORD(USINT_TO_DINT(C_Actia_Batt2_MyStatus[2])), 8)) + USINT_TO_DINT(C_Actia_Batt2_MyStatus[1])) * 0.1;
        (* Sum: '<S583>/Add' incorporates:
         *  ArithShift: '<S582>/Shift Arithmetic'
         *  Constant: '<S581>/Constant'
         *  DataTypeConversion: '<S582>/Data Type Conversion'
         *  Product: '<S583>/Product'
         *  Sum: '<S582>/Add' *)
        rtb_Add_g := DINT_TO_REAL(DWORD_TO_DINT(SHL(DINT_TO_DWORD(USINT_TO_DINT(C_LB_Batt2_Status03_Msg[1])), 8)) + USINT_TO_DINT(C_LB_Batt2_Status03_Msg[0])) * 0.1;
        (* Sum: '<S569>/Add' incorporates:
         *  ArithShift: '<S568>/Shift Arithmetic'
         *  Constant: '<S564>/Constant'
         *  DataTypeConversion: '<S568>/Data Type Conversion'
         *  Product: '<S569>/Product'
         *  Sum: '<S568>/Add' *)
        rtb_Add_ic5 := DINT_TO_REAL(DWORD_TO_DINT(SHL(DINT_TO_DWORD(USINT_TO_DINT(C_LB_Batt2_Status01_Msg[5])), 8)) + USINT_TO_DINT(C_LB_Batt2_Status01_Msg[4])) * 0.1;
        (* MultiPortSwitch: '<S761>/Multiport Switch' incorporates:
         *  Constant: '<S761>/Constant'
         *  MinMax: '<S761>/Min' *)

        CASE TRUNC(rtb_BattSelect) OF
            1: 
                (* Switch: '<S286>/Switch' incorporates:
                 *  Constant: '<S273>/Constant3'
                 *  Constant: '<S273>/SafeValue_NA '
                 *  RelationalOperator: '<S286>/GreaterThan'
                 *  Switch: '<S286>/Switch1' *)

                IF C_Actia_Batt2_MyStatus_Timeout THEN 
                    rtb_Add_h := 0.0;
                ELSIF rtb_Add_h > 6553.5 THEN 
                    (* Switch: '<S286>/Switch1' incorporates:
                     *  Constant: '<S273>/SafeValue_Error' *)
                    rtb_Add_h := 0.0;
                END_IF;

                (* End of Switch: '<S286>/Switch' *)
            2: 
                (* Switch: '<S569>/Switch' incorporates:
                 *  Constant: '<S564>/Constant3'
                 *  Constant: '<S564>/Constant4'
                 *  RelationalOperator: '<S569>/GreaterThan'
                 *  Switch: '<S569>/Switch1' *)

                IF C_LB_Batt2_Status01_Timeout THEN 
                    rtb_Add_ic5 := 0.0;
                ELSIF rtb_Add_ic5 > 6553.5 THEN 
                    (* Switch: '<S569>/Switch1' incorporates:
                     *  Constant: '<S564>/Constant4' *)
                    rtb_Add_ic5 := 0.0;
                END_IF;

                (* End of Switch: '<S569>/Switch' *)
                

                (* Switch: '<S583>/Switch' incorporates:
                 *  Constant: '<S581>/Constant3'
                 *  Constant: '<S581>/Constant4'
                 *  RelationalOperator: '<S583>/GreaterThan'
                 *  Switch: '<S583>/Switch1' *)

                IF C_LB_Batt2_Status03_Timeout THEN 
                    rtb_Add_g := 0.0;
                ELSIF rtb_Add_g > 6553.5 THEN 
                    (* Switch: '<S583>/Switch1' incorporates:
                     *  Constant: '<S581>/Constant4' *)
                    rtb_Add_g := 0.0;
                END_IF;

                (* End of Switch: '<S583>/Switch' *)
                rtb_Add_h := MIN(rtb_Add_g, rtb_Add_ic5);
            3: 
                rtb_Add_h := 0.0;
            ELSE
                rtb_Add_h := 0.0;
        END_CASE;

        (* End of MultiPortSwitch: '<S761>/Multiport Switch' *)
        

        (* Sum: '<S347>/Add' incorporates:
         *  ArithShift: '<S346>/Shift Arithmetic'
         *  Constant: '<S334>/Constant'
         *  DataTypeConversion: '<S346>/Data Type Conversion'
         *  Product: '<S347>/Product'
         *  Sum: '<S346>/Add' *)
        rtb_Add_g := DINT_TO_REAL(DWORD_TO_DINT(SHL(DINT_TO_DWORD(USINT_TO_DINT(C_Actia_Batt3_MyStatus[2])), 8)) + USINT_TO_DINT(C_Actia_Batt3_MyStatus[1])) * 0.1;
        (* Sum: '<S663>/Add' incorporates:
         *  ArithShift: '<S662>/Shift Arithmetic'
         *  Constant: '<S661>/Constant'
         *  DataTypeConversion: '<S662>/Data Type Conversion'
         *  Product: '<S663>/Product'
         *  Sum: '<S662>/Add' *)
        rtb_Add_ic5 := DINT_TO_REAL(DWORD_TO_DINT(SHL(DINT_TO_DWORD(USINT_TO_DINT(C_LB_Batt3_Status03_Msg[1])), 8)) + USINT_TO_DINT(C_LB_Batt3_Status03_Msg[0])) * 0.1;
        (* Sum: '<S649>/Add' incorporates:
         *  ArithShift: '<S648>/Shift Arithmetic'
         *  Constant: '<S644>/Constant'
         *  DataTypeConversion: '<S648>/Data Type Conversion'
         *  Product: '<S649>/Product'
         *  Sum: '<S648>/Add' *)
        rtb_Add_kf := DINT_TO_REAL(DWORD_TO_DINT(SHL(DINT_TO_DWORD(USINT_TO_DINT(C_LB_Batt3_Status01_Msg[5])), 8)) + USINT_TO_DINT(C_LB_Batt3_Status01_Msg[4])) * 0.1;
        (* MultiPortSwitch: '<S762>/Multiport Switch' incorporates:
         *  Constant: '<S762>/Constant'
         *  MinMax: '<S762>/Min' *)

        CASE TRUNC(rtb_BattSelect_i) OF
            1: 
                (* Switch: '<S347>/Switch' incorporates:
                 *  Constant: '<S334>/Constant3'
                 *  Constant: '<S334>/SafeValue_NA '
                 *  RelationalOperator: '<S347>/GreaterThan'
                 *  Switch: '<S347>/Switch1' *)

                IF C_Actia_Batt3_MyStatus_Timeout THEN 
                    rtb_Add_g := 0.0;
                ELSIF rtb_Add_g > 6553.5 THEN 
                    (* Switch: '<S347>/Switch1' incorporates:
                     *  Constant: '<S334>/SafeValue_Error' *)
                    rtb_Add_g := 0.0;
                END_IF;

                (* End of Switch: '<S347>/Switch' *)
            2: 
                (* Switch: '<S649>/Switch' incorporates:
                 *  Constant: '<S644>/Constant3'
                 *  Constant: '<S644>/Constant4'
                 *  RelationalOperator: '<S649>/GreaterThan'
                 *  Switch: '<S649>/Switch1' *)

                IF C_LB_Batt3_Status01_Timeout THEN 
                    rtb_Add_kf := 0.0;
                ELSIF rtb_Add_kf > 6553.5 THEN 
                    (* Switch: '<S649>/Switch1' incorporates:
                     *  Constant: '<S644>/Constant4' *)
                    rtb_Add_kf := 0.0;
                END_IF;

                (* End of Switch: '<S649>/Switch' *)
                

                (* Switch: '<S663>/Switch' incorporates:
                 *  Constant: '<S661>/Constant3'
                 *  Constant: '<S661>/Constant4'
                 *  RelationalOperator: '<S663>/GreaterThan'
                 *  Switch: '<S663>/Switch1' *)

                IF C_LB_Batt3_Status03_Timeout THEN 
                    rtb_Add_ic5 := 0.0;
                ELSIF rtb_Add_ic5 > 6553.5 THEN 
                    (* Switch: '<S663>/Switch1' incorporates:
                     *  Constant: '<S661>/Constant4' *)
                    rtb_Add_ic5 := 0.0;
                END_IF;

                (* End of Switch: '<S663>/Switch' *)
                rtb_Add_g := MIN(rtb_Add_ic5, rtb_Add_kf);
            3: 
                rtb_Add_g := 0.0;
            ELSE
                rtb_Add_g := 0.0;
        END_CASE;

        (* End of MultiPortSwitch: '<S762>/Multiport Switch' *)
        

        (* Sum: '<S221>/Add' incorporates:
         *  ArithShift: '<S220>/Shift Arithmetic'
         *  Constant: '<S210>/Constant'
         *  DataTypeConversion: '<S220>/Data Type Conversion'
         *  Product: '<S221>/Product'
         *  Sum: '<S220>/Add' *)
        rtb_Add_ic5 := DINT_TO_REAL(DWORD_TO_DINT(SHL(DINT_TO_DWORD(USINT_TO_DINT(C_Actia_Batt1_MyStatus[4])), 8)) + USINT_TO_DINT(C_Actia_Batt1_MyStatus[3])) * 0.1;
        (* Sum: '<S491>/Add' incorporates:
         *  ArithShift: '<S490>/Shift Arithmetic'
         *  Constant: '<S485>/Constant'
         *  DataTypeConversion: '<S490>/Data Type Conversion'
         *  Product: '<S491>/Product'
         *  Sum: '<S490>/Add' *)
        rtb_Add_kf := DINT_TO_REAL(DWORD_TO_DINT(SHL(DINT_TO_DWORD(USINT_TO_DINT(C_LB_Batt1_Status01_Msg[7])), 8)) + USINT_TO_DINT(C_LB_Batt1_Status01_Msg[6])) * 0.1;
        (* MultiPortSwitch: '<S757>/Multiport Switch' incorporates:
         *  Constant: '<S757>/Constant' *)

        CASE TRUNC(rtb_BattSelect_f) OF
            1: 
                (* Switch: '<S221>/Switch' incorporates:
                 *  Constant: '<S210>/Constant3'
                 *  Constant: '<S210>/SafeValue_NA '
                 *  RelationalOperator: '<S221>/GreaterThan'
                 *  Switch: '<S221>/Switch1' *)

                IF C_Actia_Batt1_MyStatus_Timeout THEN 
                    rtb_Add_ic5 := 0.0;
                ELSIF rtb_Add_ic5 > 6553.5 THEN 
                    (* Switch: '<S221>/Switch1' incorporates:
                     *  Constant: '<S210>/SafeValue_Error' *)
                    rtb_Add_ic5 := 0.0;
                END_IF;

                (* End of Switch: '<S221>/Switch' *)
            2: 
                (* Switch: '<S491>/Switch' incorporates:
                 *  Constant: '<S485>/Constant3'
                 *  Constant: '<S485>/Constant4'
                 *  RelationalOperator: '<S491>/GreaterThan'
                 *  Switch: '<S491>/Switch1' *)

                IF C_LB_Batt1_Status01_Timeout THEN 
                    rtb_Add_ic5 := 0.0;
                ELSIF rtb_Add_kf > 6553.5 THEN 
                    (* Switch: '<S491>/Switch1' incorporates:
                     *  Constant: '<S485>/Constant4' *)
                    rtb_Add_ic5 := 0.0;
                ELSE 
                    (* Switch: '<S491>/Switch1' *)
                    rtb_Add_ic5 := rtb_Add_kf;
                END_IF;

                (* End of Switch: '<S491>/Switch' *)
            3: 
                rtb_Add_ic5 := 0.0;
            ELSE
                rtb_Add_ic5 := 0.0;
        END_CASE;

        (* End of MultiPortSwitch: '<S757>/Multiport Switch' *)
        

        (* Sum: '<S282>/Add' incorporates:
         *  ArithShift: '<S281>/Shift Arithmetic'
         *  Constant: '<S271>/Constant'
         *  DataTypeConversion: '<S281>/Data Type Conversion'
         *  Product: '<S282>/Product'
         *  Sum: '<S281>/Add' *)
        rtb_Add_kf := DINT_TO_REAL(DWORD_TO_DINT(SHL(DINT_TO_DWORD(USINT_TO_DINT(C_Actia_Batt2_MyStatus[4])), 8)) + USINT_TO_DINT(C_Actia_Batt2_MyStatus[3])) * 0.1;
        (* Sum: '<S571>/Add' incorporates:
         *  ArithShift: '<S570>/Shift Arithmetic'
         *  Constant: '<S565>/Constant'
         *  DataTypeConversion: '<S570>/Data Type Conversion'
         *  Product: '<S571>/Product'
         *  Sum: '<S570>/Add' *)
        rtb_Add_j3 := DINT_TO_REAL(DWORD_TO_DINT(SHL(DINT_TO_DWORD(USINT_TO_DINT(C_LB_Batt2_Status01_Msg[7])), 8)) + USINT_TO_DINT(C_LB_Batt2_Status01_Msg[6])) * 0.1;
        (* MultiPortSwitch: '<S758>/Multiport Switch' incorporates:
         *  Constant: '<S758>/Constant' *)

        CASE TRUNC(rtb_BattSelect) OF
            1: 
                (* Switch: '<S282>/Switch' incorporates:
                 *  Constant: '<S271>/Constant3'
                 *  Constant: '<S271>/SafeValue_NA '
                 *  RelationalOperator: '<S282>/GreaterThan'
                 *  Switch: '<S282>/Switch1' *)

                IF C_Actia_Batt2_MyStatus_Timeout THEN 
                    rtb_Add_kf := 0.0;
                ELSIF rtb_Add_kf > 6553.5 THEN 
                    (* Switch: '<S282>/Switch1' incorporates:
                     *  Constant: '<S271>/SafeValue_Error' *)
                    rtb_Add_kf := 0.0;
                END_IF;

                (* End of Switch: '<S282>/Switch' *)
            2: 
                (* Switch: '<S571>/Switch' incorporates:
                 *  Constant: '<S565>/Constant3'
                 *  Constant: '<S565>/Constant4'
                 *  RelationalOperator: '<S571>/GreaterThan'
                 *  Switch: '<S571>/Switch1' *)

                IF C_LB_Batt2_Status01_Timeout THEN 
                    rtb_Add_kf := 0.0;
                ELSIF rtb_Add_j3 > 6553.5 THEN 
                    (* Switch: '<S571>/Switch1' incorporates:
                     *  Constant: '<S565>/Constant4' *)
                    rtb_Add_kf := 0.0;
                ELSE 
                    (* Switch: '<S571>/Switch1' *)
                    rtb_Add_kf := rtb_Add_j3;
                END_IF;

                (* End of Switch: '<S571>/Switch' *)
            3: 
                rtb_Add_kf := 0.0;
            ELSE
                rtb_Add_kf := 0.0;
        END_CASE;

        (* End of MultiPortSwitch: '<S758>/Multiport Switch' *)
        

        (* Sum: '<S343>/Add' incorporates:
         *  ArithShift: '<S342>/Shift Arithmetic'
         *  Constant: '<S332>/Constant'
         *  DataTypeConversion: '<S342>/Data Type Conversion'
         *  Product: '<S343>/Product'
         *  Sum: '<S342>/Add' *)
        rtb_Add_j3 := DINT_TO_REAL(DWORD_TO_DINT(SHL(DINT_TO_DWORD(USINT_TO_DINT(C_Actia_Batt3_MyStatus[4])), 8)) + USINT_TO_DINT(C_Actia_Batt3_MyStatus[3])) * 0.1;
        (* Sum: '<S651>/Add' incorporates:
         *  ArithShift: '<S650>/Shift Arithmetic'
         *  Constant: '<S645>/Constant'
         *  DataTypeConversion: '<S650>/Data Type Conversion'
         *  Product: '<S651>/Product'
         *  Sum: '<S650>/Add' *)
        rtb_Add_cv := DINT_TO_REAL(DWORD_TO_DINT(SHL(DINT_TO_DWORD(USINT_TO_DINT(C_LB_Batt3_Status01_Msg[7])), 8)) + USINT_TO_DINT(C_LB_Batt3_Status01_Msg[6])) * 0.1;
        (* MultiPortSwitch: '<S759>/Multiport Switch' incorporates:
         *  Constant: '<S759>/Constant' *)

        CASE TRUNC(rtb_BattSelect_i) OF
            1: 
                (* Switch: '<S343>/Switch' incorporates:
                 *  Constant: '<S332>/Constant3'
                 *  Constant: '<S332>/SafeValue_NA '
                 *  RelationalOperator: '<S343>/GreaterThan'
                 *  Switch: '<S343>/Switch1' *)

                IF C_Actia_Batt3_MyStatus_Timeout THEN 
                    rtb_Add_j3 := 0.0;
                ELSIF rtb_Add_j3 > 6553.5 THEN 
                    (* Switch: '<S343>/Switch1' incorporates:
                     *  Constant: '<S332>/SafeValue_Error' *)
                    rtb_Add_j3 := 0.0;
                END_IF;

                (* End of Switch: '<S343>/Switch' *)
            2: 
                (* Switch: '<S651>/Switch' incorporates:
                 *  Constant: '<S645>/Constant3'
                 *  Constant: '<S645>/Constant4'
                 *  RelationalOperator: '<S651>/GreaterThan'
                 *  Switch: '<S651>/Switch1' *)

                IF C_LB_Batt3_Status01_Timeout THEN 
                    rtb_Add_j3 := 0.0;
                ELSIF rtb_Add_cv > 6553.5 THEN 
                    (* Switch: '<S651>/Switch1' incorporates:
                     *  Constant: '<S645>/Constant4' *)
                    rtb_Add_j3 := 0.0;
                ELSE 
                    (* Switch: '<S651>/Switch1' *)
                    rtb_Add_j3 := rtb_Add_cv;
                END_IF;

                (* End of Switch: '<S651>/Switch' *)
            3: 
                rtb_Add_j3 := 0.0;
            ELSE
                rtb_Add_j3 := 0.0;
        END_CASE;

        (* End of MultiPortSwitch: '<S759>/Multiport Switch' *)
        

        (* Sum: '<S247>/Add' incorporates:
         *  Constant: '<S243>/Constant'
         *  Product: '<S247>/Product' *)
        rtb_Add_cv := USINT_TO_REAL(C_Actia_Batt1_ADS_8[5]) * 5.0;
        (* Sum: '<S467>/Add' incorporates:
         *  ArithShift: '<S466>/Shift Arithmetic'
         *  DataTypeConversion: '<S466>/Data Type Conversion'
         *  Sum: '<S466>/Add' *)
        rtb_Add_ci := DINT_TO_REAL(DWORD_TO_DINT(SHL(DINT_TO_DWORD(USINT_TO_DINT(C_LB_Batt1_InsulationMonitor_Msg[1])), 8)) + USINT_TO_DINT(C_LB_Batt1_InsulationMonitor_Msg[0]));
        (* Switch: '<S467>/Switch' incorporates:
         *  Constant: '<S463>/Constant4' *)

        IF C_LB_Batt1_InsulationMonitor_Timeout THEN 
            rtb_Add_ci := 0.0;
        END_IF;

        (* End of Switch: '<S467>/Switch' *)
        

        (* Sum: '<S732>/Subtract' incorporates:
         *  Constant: '<S732>/Constant4'
         *  Gain: '<S732>/mV to V' *)
        rtb_Add_ci := (0.001 * rtb_Add_ci) - 2.48;
        (* MultiPortSwitch: '<S729>/Multiport Switch' incorporates:
         *  Abs: '<S732>/Abs'
         *  Constant: '<S729>/Constant'
         *  Constant: '<S732>/Constant1'
         *  Constant: '<S732>/Constant2'
         *  Product: '<S732>/Divide'
         *  Product: '<S732>/Product'
         *  Sum: '<S732>/Subtract1' *)

        CASE TRUNC(rtb_BattSelect_f) OF
            1: 
                (* Switch: '<S247>/Switch' incorporates:
                 *  Constant: '<S243>/Constant3'
                 *  Constant: '<S243>/SafeValue_NA '
                 *  RelationalOperator: '<S247>/GreaterThan'
                 *  Switch: '<S247>/Switch1' *)

                IF C_Actia_Batt1_ADS_8_Timeout THEN 
                    rtb_Add_cv := 0.0;
                ELSIF rtb_Add_cv > 0.0 THEN 
                    (* Switch: '<S247>/Switch1' incorporates:
                     *  Constant: '<S243>/SafeValue_Error' *)
                    rtb_Add_cv := 0.0;
                END_IF;

                (* End of Switch: '<S247>/Switch' *)
            2: 
                rtb_Add_cv := ((rtb_Add_psl * 10.0) / ABS(rtb_Add_ci)) - 2000.0;
            3: 
                rtb_Add_cv := 0.0;
            ELSE
                rtb_Add_cv := 0.0;
        END_CASE;

